LIN {X 0,Y 483.162,Z 602.716,A -85,B 0,C 180,E1 -6752.605,E2 -6752.605} C_VEL
LIN {X 0,Y 482.874,Z 611.081,A -85,B 0,C 180,E1 -6753.546,E2 -6753.546} C_VEL
LIN {X 0,Y 482.488,Z 618.843,A -85,B 0,C 180,E1 -6754.594,E2 -6754.594} C_VEL
LIN {X 0,Y 482.235,Z 626.404,A -85,B 0,C 180,E1 -6755.854,E2 -6755.854} C_VEL
LIN {X 0,Y 481.962,Z 632.514,A -85,B 0,C 180,E1 -6757.125,E2 -6757.125} C_VEL
LIN {X 0,Y 481.753,Z 637.329,A -85,B 0,C 180,E1 -6758.388,E2 -6758.388} C_VEL
LIN {X 0,Y 481.542,Z 641.081,A -85,B 0,C 180,E1 -6759.661,E2 -6759.661} C_VEL
LIN {X 0,Y 481.419,Z 643.812,A -85,B 0,C 180,E1 -6760.939,E2 -6760.939} C_VEL
LIN {X 0,Y 481.414,Z 645.378,A -85,B 0,C 180,E1 -6762.012,E2 -6762.012} C_VEL
LIN {X 0,Y 481.342,Z 646.455,A -85,B 0,C 180,E1 -6763.509,E2 -6763.509} C_VEL
LIN {X 0,Y 481.387,Z 646.173,A -85,B 0,C 180,E1 -6765.235,E2 -6765.235} C_VEL
LIN {X 0,Y 481.377,Z 645.433,A -85,B 0,C 180,E1 -6766.104,E2 -6766.104} C_VEL
LIN {X 0,Y 481.429,Z 644.224,A -85,B 0,C 180,E1 -6766.975,E2 -6766.975} C_VEL
LIN {X 0,Y 481.589,Z 641.181,A -85,B 0,C 180,E1 -6768.457,E2 -6768.457} C_VEL
LIN {X 0,Y 481.792,Z 636.402,A -85,B 0,C 180,E1 -6770.047,E2 -6770.047} C_VEL
LIN {X 0,Y 482.078,Z 631.006,A -85,B 0,C 180,E1 -6771.374,E2 -6771.374} C_VEL
LIN {X 0,Y 482.374,Z 624.124,A -85,B 0,C 180,E1 -6772.711,E2 -6772.711} C_VEL
LIN {X 0,Y 482.765,Z 616.715,A -85,B 0,C 180,E1 -6773.867,E2 -6773.867} C_VEL
LIN {X 0,Y 483.101,Z 608.237,A -85,B 0,C 180,E1 -6774.952,E2 -6774.952} C_VEL
LIN {X 0,Y 483.452,Z 598.406,A -85,B 0,C 180,E1 -6775.971,E2 -6775.971} C_VEL
LIN {X 0,Y 483.892,Z 587.565,A -85,B 0,C 180,E1 -6776.871,E2 -6776.871} C_VEL
LIN {X 0,Y 484.235,Z 576.341,A -85,B 0,C 180,E1 -6777.61,E2 -6777.61} C_VEL
LIN {X 0,Y 484.067,Z 572.549,A -85,B 0,C 180,E1 -6777.827,E2 -6777.827} C_VEL
LIN {X 0,Y 481.719,Z 564.483,A -85,B 0,C 180,E1 -6778.333,E2 -6778.333} C_VEL
LIN {X 0,Y 481.643,Z 564.489,A -85,B 0,C 180,E1 -6781.687,E2 -6781.687} C_VEL
LIN {X 0,Y 481.685,Z 564.485,A -85,B 0,C 180,E1 -6784.681,E2 -6784.681} C_VEL
LIN {X 0,Y 481.655,Z 564.49,A -85,B 0,C 180,E1 -6788.008,E2 -6788.008} C_VEL
LIN {X 0,Y 481.76,Z 564.652,A -85,B 0,C 180,E1 -6790.063,E2 -6790.063} C_VEL
LIN {X 0,Y 482.299,Z 569.987,A -85,B 0,C 180,E1 -6792.089,E2 -6792.089} C_VEL
LIN {X 0,Y 482.189,Z 577.722,A -85,B 0,C 180,E1 -6795.018,E2 -6795.018} C_VEL
LIN {X 0,Y 482.112,Z 585.89,A -85,B 0,C 180,E1 -6798.025,E2 -6798.025} C_VEL
LIN {X 0,Y 481.911,Z 594.241,A -85,B 0,C 180,E1 -6801.164,E2 -6801.164} C_VEL
LIN {X 0,Y 481.765,Z 602.576,A -85,B 0,C 180,E1 -6804.302,E2 -6804.302} C_VEL
LIN {X 0,Y 481.644,Z 610.581,A -85,B 0,C 180,E1 -6807.324,E2 -6807.324} C_VEL
LIN {X 0,Y 481.461,Z 618.342,A -85,B 0,C 180,E1 -6810.244,E2 -6810.244} C_VEL
LIN {X 0,Y 481.363,Z 623.373,A -85,B 0,C 180,E1 -6812.133,E2 -6812.133} C_VEL
LIN {X 0,Y 483.918,Z 637.058,A -85,B 0,C 180,E1 -6812.586,E2 -6812.586} C_VEL
LIN {X 0,Y 483.654,Z 649.638,A -85,B 0,C 180,E1 -6813.085,E2 -6813.085} C_VEL
LIN {X 0,Y 483.238,Z 662.401,A -85,B 0,C 180,E1 -6813.784,E2 -6813.784} C_VEL
LIN {X 0,Y 482.867,Z 673.508,A -85,B 0,C 180,E1 -6814.571,E2 -6814.571} C_VEL
LIN {X 0,Y 482.439,Z 683.68,A -85,B 0,C 180,E1 -6815.47,E2 -6815.47} C_VEL
LIN {X 0,Y 482.016,Z 694.049,A -85,B 0,C 180,E1 -6816.613,E2 -6816.613} C_VEL
LIN {X 0,Y 481.645,Z 702.132,A -85,B 0,C 180,E1 -6817.705,E2 -6817.705} C_VEL
LIN {X 0,Y 481.37,Z 709.469,A -85,B 0,C 180,E1 -6818.921,E2 -6818.921} C_VEL
LIN {X 0,Y 481.161,Z 716.363,A -85,B 0,C 180,E1 -6820.37,E2 -6820.37} C_VEL
LIN {X 0,Y 480.998,Z 721.451,A -85,B 0,C 180,E1 -6821.752,E2 -6821.752} C_VEL
LIN {X 0,Y 480.857,Z 724.91,A -85,B 0,C 180,E1 -6823.004,E2 -6823.004} C_VEL
LIN {X 0,Y 480.806,Z 726.732,A -85,B 0,C 180,E1 -6823.876,E2 -6823.876} C_VEL
LIN {X 0,Y 480.797,Z 728.085,A -85,B 0,C 180,E1 -6824.746,E2 -6824.746} C_VEL
LIN {X 0,Y 480.787,Z 729.027,A -85,B 0,C 180,E1 -6825.612,E2 -6825.612} C_VEL
LIN {X 0,Y 480.739,Z 729.53,A -85,B 0,C 180,E1 -6826.473,E2 -6826.473} C_VEL
LIN {X 0,Y 480.756,Z 729.594,A -85,B 0,C 180,E1 -6827.334,E2 -6827.334} C_VEL
LIN {X 0,Y 480.841,Z 729.198,A -85,B 0,C 180,E1 -6828.309,E2 -6828.309} C_VEL
LIN {X 0,Y 480.833,Z 727.348,A -85,B 0,C 180,E1 -6829.899,E2 -6829.899} C_VEL
LIN {X 0,Y 480.909,Z 724.804,A -85,B 0,C 180,E1 -6831.174,E2 -6831.174} C_VEL
LIN {X 0,Y 481.041,Z 721.245,A -85,B 0,C 180,E1 -6832.445,E2 -6832.445} C_VEL
LIN {X 0,Y 481.163,Z 715.912,A -85,B 0,C 180,E1 -6833.873,E2 -6833.873} C_VEL
LIN {X 0,Y 481.336,Z 709.617,A -85,B 0,C 180,E1 -6835.184,E2 -6835.184} C_VEL
LIN {X 0,Y 481.658,Z 701.976,A -85,B 0,C 180,E1 -6836.445,E2 -6836.445} C_VEL
LIN {X 0,Y 482.063,Z 692.502,A -85,B 0,C 180,E1 -6837.703,E2 -6837.703} C_VEL
LIN {X 0,Y 482.511,Z 682.637,A -85,B 0,C 180,E1 -6838.748,E2 -6838.748} C_VEL
LIN {X 0,Y 482.943,Z 671.629,A -85,B 0,C 180,E1 -6839.688,E2 -6839.688} C_VEL
LIN {X 0,Y 483.344,Z 660.923,A -85,B 0,C 180,E1 -6840.417,E2 -6840.417} C_VEL
LIN {X 0,Y 483.769,Z 649.032,A -85,B 0,C 180,E1 -6841.041,E2 -6841.041} C_VEL
LIN {X 0,Y 483.89,Z 636.377,A -85,B 0,C 180,E1 -6841.535,E2 -6841.535} C_VEL
LIN {X 0,Y 481.718,Z 625.568,A -85,B 0,C 180,E1 -6841.895,E2 -6841.895} C_VEL
LIN {X 0,Y 481.47,Z 624.18,A -85,B 0,C 180,E1 -6841.935,E2 -6841.935} C_VEL
LIN {X 0,Y 481.677,Z 615.891,A -85,B 0,C 180,E1 -6845.023,E2 -6845.023} C_VEL
LIN {X 0,Y 481.773,Z 606.79,A -85,B 0,C 180,E1 -6848.388,E2 -6848.388} C_VEL
LIN {X 0,Y 481.871,Z 599.852,A -85,B 0,C 180,E1 -6850.93,E2 -6850.93} C_VEL
LIN {X 0,Y 481.991,Z 592.674,A -85,B 0,C 180,E1 -6853.492,E2 -6853.492} C_VEL
LIN {X 0,Y 482.013,Z 583.839,A -85,B 0,C 180,E1 -6856.519,E2 -6856.519} C_VEL
LIN {X 0,Y 482.005,Z 574.554,A -85,B 0,C 180,E1 -6859.595,E2 -6859.595} C_VEL
LIN {X 0,Y 481.898,Z 566.032,A -85,B 0,C 180,E1 -6862.283,E2 -6862.283} C_VEL
LIN {X 0,Y 481.683,Z 564.488,A -85,B 0,C 180,E1 -6862.802,E2 -6862.802} C_VEL
LIN {X 0,Y 481.7,Z 564.488,A -85,B 0,C 180,E1 -6865.958,E2 -6865.958} C_VEL
LIN {X 0,Y 481.701,Z 564.485,A -85,B 0,C 180,E1 -6868.782,E2 -6868.782} C_VEL
LIN {X 0,Y 481.654,Z 564.492,A -85,B 0,C 180,E1 -6872.191,E2 -6872.191} C_VEL
LIN {X 0,Y 481.688,Z 564.487,A -85,B 0,C 180,E1 -6874.683,E2 -6874.683} C_VEL
LIN {X 0,Y 481.654,Z 564.49,A -85,B 0,C 180,E1 -6878.009,E2 -6878.009} C_VEL
LIN {X 0,Y 481.681,Z 564.488,A -85,B 0,C 180,E1 -6880.651,E2 -6880.651} C_VEL
LIN {X 0,Y 481.68,Z 564.487,A -85,B 0,C 180,E1 -6883.296,E2 -6883.296} C_VEL
LIN {X 0,Y 481.686,Z 564.486,A -85,B 0,C 180,E1 -6886.847,E2 -6886.847} C_VEL
LIN {X 0,Y 481.741,Z 564.602,A -85,B 0,C 180,E1 -6889.871,E2 -6889.871} C_VEL
LIN {X 0,Y 483.91,Z 575.619,A -85,B 0,C 180,E1 -6893.015,E2 -6893.015} C_VEL
LIN {X 0,Y 484.216,Z 579.325,A -85,B 0,C 180,E1 -6893.99,E2 -6893.99} C_VEL
LIN {X 0,Y 483.665,Z 591.413,A -85,B 0,C 180,E1 -6896.984,E2 -6896.984} C_VEL
LIN {X 0,Y 483.156,Z 605.658,A -85,B 0,C 180,E1 -6900.36,E2 -6900.36} C_VEL
LIN {X 0,Y 482.7,Z 620.019,A -85,B 0,C 180,E1 -6903.637,E2 -6903.637} C_VEL
LIN {X 0,Y 482.294,Z 634.452,A -85,B 0,C 180,E1 -6906.832,E2 -6906.832} C_VEL
LIN {X 0,Y 481.964,Z 648.924,A -85,B 0,C 180,E1 -6909.961,E2 -6909.961} C_VEL
LIN {X 0,Y 481.681,Z 663.387,A -85,B 0,C 180,E1 -6913.035,E2 -6913.035} C_VEL
LIN {X 0,Y 481.527,Z 672.733,A -85,B 0,C 180,E1 -6915.013,E2 -6915.013} C_VEL
LIN {X 0,Y 482.885,Z 686.464,A -85,B 0,C 180,E1 -6915.368,E2 -6915.368} C_VEL
LIN {X 0,Y 483.795,Z 694.327,A -85,B 0,C 180,E1 -6915.65,E2 -6915.65} C_VEL
LIN {X 0,Y 483.332,Z 706.466,A -85,B 0,C 180,E1 -6916.173,E2 -6916.173} C_VEL
LIN {X 0,Y 482.877,Z 718.803,A -85,B 0,C 180,E1 -6916.888,E2 -6916.888} C_VEL
LIN {X 0,Y 482.506,Z 729.607,A -85,B 0,C 180,E1 -6917.685,E2 -6917.685} C_VEL
LIN {X 0,Y 482.04,Z 740.179,A -85,B 0,C 180,E1 -6918.649,E2 -6918.649} C_VEL
LIN {X 0,Y 481.684,Z 749.542,A -85,B 0,C 180,E1 -6919.705,E2 -6919.705} C_VEL
LIN {X 0,Y 481.423,Z 758.694,A -85,B 0,C 180,E1 -6920.972,E2 -6920.972} C_VEL
LIN {X 0,Y 481.209,Z 766.056,A -85,B 0,C 180,E1 -6922.237,E2 -6922.237} C_VEL
LIN {X 0,Y 481.063,Z 772.846,A -85,B 0,C 180,E1 -6923.712,E2 -6923.712} C_VEL
LIN {X 0,Y 481.013,Z 777.288,A -85,B 0,C 180,E1 -6924.972,E2 -6924.972} C_VEL
LIN {X 0,Y 480.986,Z 779.659,A -85,B 0,C 180,E1 -6925.811,E2 -6925.811} C_VEL
LIN {X 0,Y 480.985,Z 781.572,A -85,B 0,C 180,E1 -6926.65,E2 -6926.65} C_VEL
LIN {X 0,Y 480.949,Z 783.04,A -85,B 0,C 180,E1 -6927.488,E2 -6927.488} C_VEL
LIN {X 0,Y 480.93,Z 784.074,A -85,B 0,C 180,E1 -6928.326,E2 -6928.326} C_VEL
LIN {X 0,Y 480.898,Z 784.693,A -85,B 0,C 180,E1 -6929.163,E2 -6929.163} C_VEL
LIN {X 0,Y 480.892,Z 784.904,A -85,B 0,C 180,E1 -6930.001,E2 -6930.001} C_VEL
LIN {X 0,Y 480.898,Z 784.69,A -85,B 0,C 180,E1 -6930.838,E2 -6930.838} C_VEL
LIN {X 0,Y 480.932,Z 784.059,A -85,B 0,C 180,E1 -6931.676,E2 -6931.676} C_VEL
LIN {X 0,Y 480.952,Z 783.019,A -85,B 0,C 180,E1 -6932.513,E2 -6932.513} C_VEL
LIN {X 0,Y 480.986,Z 781.569,A -85,B 0,C 180,E1 -6933.351,E2 -6933.351} C_VEL
LIN {X 0,Y 480.975,Z 778.572,A -85,B 0,C 180,E1 -6934.61,E2 -6934.61} C_VEL
LIN {X 0,Y 481.087,Z 774.505,A -85,B 0,C 180,E1 -6935.87,E2 -6935.87} C_VEL
LIN {X 0,Y 481.154,Z 768.267,A -85,B 0,C 180,E1 -6937.344,E2 -6937.344} C_VEL
LIN {X 0,Y 481.364,Z 761.397,A -85,B 0,C 180,E1 -6938.607,E2 -6938.607} C_VEL
LIN {X 0,Y 481.576,Z 752.955,A -85,B 0,C 180,E1 -6939.874,E2 -6939.874} C_VEL
LIN {X 0,Y 481.917,Z 744.301,A -85,B 0,C 180,E1 -6940.929,E2 -6940.929} C_VEL
LIN {X 0,Y 482.396,Z 733.747,A -85,B 0,C 180,E1 -6941.974,E2 -6941.974} C_VEL
LIN {X 0,Y 482.702,Z 723.405,A -85,B 0,C 180,E1 -6942.808,E2 -6942.808} C_VEL
LIN {X 0,Y 483.164,Z 711.61,A -85,B 0,C 180,E1 -6943.566,E2 -6943.566} C_VEL
LIN {X 0,Y 483.566,Z 699.818,A -85,B 0,C 180,E1 -6944.144,E2 -6944.144} C_VEL
LIN {X 0,Y 483.631,Z 691.789,A -85,B 0,C 180,E1 -6944.451,E2 -6944.451} C_VEL
LIN {X 0,Y 482.182,Z 680.276,A -85,B 0,C 180,E1 -6944.819,E2 -6944.819} C_VEL
LIN {X 0,Y 481.535,Z 673.024,A -85,B 0,C 180,E1 -6944.988,E2 -6944.988} C_VEL
LIN {X 0,Y 481.833,Z 657.99,A -85,B 0,C 180,E1 -6948.193,E2 -6948.193} C_VEL
LIN {X 0,Y 482.121,Z 643.287,A -85,B 0,C 180,E1 -6951.373,E2 -6951.373} C_VEL
LIN {X 0,Y 482.454,Z 629.918,A -85,B 0,C 180,E1 -6954.301,E2 -6954.301} C_VEL
LIN {X 0,Y 482.857,Z 616.074,A -85,B 0,C 180,E1 -6957.394,E2 -6957.394} C_VEL
LIN {X 0,Y 483.243,Z 603.092,A -85,B 0,C 180,E1 -6960.357,E2 -6960.357} C_VEL
LIN {X 0,Y 483.675,Z 590.668,A -85,B 0,C 180,E1 -6963.266,E2 -6963.266} C_VEL
LIN {X 0,Y 484.095,Z 578.209,A -85,B 0,C 180,E1 -6966.271,E2 -6966.271} C_VEL
LIN {X 0,Y 483.339,Z 572.934,A -85,B 0,C 180,E1 -6967.641,E2 -6967.641} C_VEL
LIN {X 0,Y 481.704,Z 564.485,A -85,B 0,C 180,E1 -6969.938,E2 -6969.938} C_VEL
LIN {X 0,Y 481.644,Z 564.493,A -85,B 0,C 180,E1 -6973.3,E2 -6973.3} C_VEL
LIN {X 0,Y 481.663,Z 564.49,A -85,B 0,C 180,E1 -6975.641,E2 -6975.641} C_VEL
LIN {X 0,Y 481.661,Z 564.49,A -85,B 0,C 180,E1 -6978.958,E2 -6978.958} C_VEL
LIN {X 0,Y 481.66,Z 564.489,A -85,B 0,C 180,E1 -6981.993,E2 -6981.993} C_VEL
LIN {X 0,Y 481.698,Z 564.483,A -85,B 0,C 180,E1 -6985.318,E2 -6985.318} C_VEL
LIN {X 0,Y 481.649,Z 564.492,A -85,B 0,C 180,E1 -6988.312,E2 -6988.312} C_VEL
LIN {X 0,Y 481.705,Z 564.481,A -85,B 0,C 180,E1 -6991.219,E2 -6991.219} C_VEL
LIN {X 0,Y 481.705,Z 564.483,A -85,B 0,C 180,E1 -6994.043,E2 -6994.043} C_VEL
LIN {X 0,Y 481.679,Z 564.486,A -85,B 0,C 180,E1 -6996.812,E2 -6996.812} C_VEL
LIN {X 0,Y 481.7,Z 564.482,A -85,B 0,C 180,E1 -6999.503,E2 -6999.503} C_VEL
LIN {X 0,Y 481.712,Z 564.483,A -85,B 0,C 180,E1 -7002.158,E2 -7002.158} C_VEL
LIN {X 0,Y 481.747,Z 564.479,A -85,B 0,C 180,E1 -7004.776,E2 -7004.776} C_VEL
LIN {X 0,Y 481.755,Z 564.478,A -85,B 0,C 180,E1 -7008.215,E2 -7008.215} C_VEL
LIN {X 0,Y 481.767,Z 564.474,A -85,B 0,C 180,E1 -7011.611,E2 -7011.611} C_VEL
LIN {X 0,Y 481.82,Z 564.47,A -85,B 0,C 180,E1 -7014.139,E2 -7014.139} C_VEL
LIN {X 0,Y 481.93,Z 564.454,A -85,B 0,C 180,E1 -7017.492,E2 -7017.492} C_VEL
LIN {X 0,Y 481.91,Z 564.459,A -85,B 0,C 180,E1 -7020.835,E2 -7020.835} C_VEL
LIN {X 0,Y 481.93,Z 564.456,A -85,B 0,C 180,E1 -7022.507,E2 -7022.507} C_VEL
LIN {X 0,Y 481.82,Z 564.469,A -85,B 0,C 180,E1 -7025.86,E2 -7025.86} C_VEL
LIN {X 0,Y 481.766,Z 564.477,A -85,B 0,C 180,E1 -7028.388,E2 -7028.388} C_VEL
LIN {X 0,Y 481.754,Z 564.477,A -85,B 0,C 180,E1 -7031.784,E2 -7031.784} C_VEL
LIN {X 0,Y 481.746,Z 564.478,A -85,B 0,C 180,E1 -7035.224,E2 -7035.224} C_VEL
LIN {X 0,Y 481.715,Z 564.483,A -85,B 0,C 180,E1 -7038.721,E2 -7038.721} C_VEL
LIN {X 0,Y 481.649,Z 564.489,A -85,B 0,C 180,E1 -7041.394,E2 -7041.394} C_VEL
LIN {X 0,Y 481.68,Z 564.486,A -85,B 0,C 180,E1 -7044.113,E2 -7044.113} C_VEL
LIN {X 0,Y 481.749,Z 564.476,A -85,B 0,C 180,E1 -7047.139,E2 -7047.139} C_VEL
LIN {X 0,Y 481.681,Z 564.485,A -85,B 0,C 180,E1 -7049.741,E2 -7049.741} C_VEL
LIN {X 0,Y 481.674,Z 564.489,A -85,B 0,C 180,E1 -7052.674,E2 -7052.674} C_VEL
LIN {X 0,Y 481.645,Z 564.489,A -85,B 0,C 180,E1 -7055.708,E2 -7055.708} C_VEL
LIN {X 0,Y 481.673,Z 564.487,A -85,B 0,C 180,E1 -7058.858,E2 -7058.858} C_VEL
LIN {X 0,Y 481.664,Z 564.487,A -85,B 0,C 180,E1 -7061.914,E2 -7061.914} C_VEL
LIN {X 0,Y 481.661,Z 564.491,A -85,B 0,C 180,E1 -7064.457,E2 -7064.457} C_VEL
LIN {X 0,Y 481.655,Z 564.489,A -85,B 0,C 180,E1 -7067.839,E2 -7067.839} C_VEL
LIN {X 0,Y 481.682,Z 564.487,A -85,B 0,C 180,E1 -7070.65,E2 -7070.65} C_VEL
LIN {X 0,Y 481.628,Z 564.492,A -85,B 0,C 180,E1 -7073.376,E2 -7073.376} C_VEL
LIN {X 0,Y 481.71,Z 564.484,A -85,B 0,C 180,E1 -7076.329,E2 -7076.329} C_VEL
LIN {X 0,Y 481.652,Z 564.489,A -85,B 0,C 180,E1 -7079.417,E2 -7079.417} C_VEL
LIN {X 0,Y 481.701,Z 564.485,A -85,B 0,C 180,E1 -7082.167,E2 -7082.167} C_VEL
LIN {X 0,Y 481.719,Z 564.482,A -85,B 0,C 180,E1 -7084.969,E2 -7084.969} C_VEL
LIN {X 0,Y 481.637,Z 564.49,A -85,B 0,C 180,E1 -7087.981,E2 -7087.981} C_VEL
LIN {X 0,Y 480.97,Z 564.576,A -85,B 0,C 180,E1 -7088.679,E2 -7088.679} C_VEL
LIN {X 0,Y 478.142,Z 564.925,A -85,B 0,C 180,E1 -7089.813,E2 -7089.813} C_VEL
LIN {X 0,Y 475.757,Z 565.225,A -85,B 0,C 180,E1 -7090.727,E2 -7090.727} C_VEL
LIN {X 0,Y 474.737,Z 565.35,A -85,B 0,C 180,E1 -7091.433,E2 -7091.433} C_VEL
LIN {X 0,Y 474.655,Z 565.36,A -85,B 0,C 180,E1 -7091.672,E2 -7091.672} C_VEL
LIN {X 0,Y 474.7,Z 565.357,A -85,B 0,C 180,E1 -7094.544,E2 -7094.544} C_VEL
LIN {X 0,Y 474.739,Z 565.35,A -85,B 0,C 180,E1 -7098.038,E2 -7098.038} C_VEL
LIN {X 0,Y 474.727,Z 565.352,A -85,B 0,C 180,E1 -7101.486,E2 -7101.486} C_VEL
LIN {X 0,Y 474.779,Z 565.346,A -85,B 0,C 180,E1 -7104.052,E2 -7104.052} C_VEL
LIN {X 0,Y 474.895,Z 565.333,A -85,B 0,C 180,E1 -7107.455,E2 -7107.455} C_VEL
LIN {X 0,Y 474.898,Z 565.381,A -85,B 0,C 180,E1 -7109.655,E2 -7109.655} C_VEL
LIN {X 0,Y 477.267,Z 574.753,A -85,B 0,C 180,E1 -7110.21,E2 -7110.21} C_VEL
LIN {X 0,Y 477.003,Z 586.419,A -85,B 0,C 180,E1 -7110.949,E2 -7110.949} C_VEL
LIN {X 0,Y 476.584,Z 596.917,A -85,B 0,C 180,E1 -7111.795,E2 -7111.795} C_VEL
LIN {X 0,Y 476.161,Z 606.491,A -85,B 0,C 180,E1 -7112.749,E2 -7112.749} C_VEL
LIN {X 0,Y 475.822,Z 615.19,A -85,B 0,C 180,E1 -7113.81,E2 -7113.81} C_VEL
LIN {X 0,Y 475.431,Z 623.719,A -85,B 0,C 180,E1 -7115.088,E2 -7115.088} C_VEL
LIN {X 0,Y 475.143,Z 630.521,A -85,B 0,C 180,E1 -7116.368,E2 -7116.368} C_VEL
LIN {X 0,Y 474.878,Z 635.986,A -85,B 0,C 180,E1 -7117.653,E2 -7117.653} C_VEL
LIN {X 0,Y 474.648,Z 640.29,A -85,B 0,C 180,E1 -7118.943,E2 -7118.943} C_VEL
LIN {X 0,Y 474.476,Z 643.537,A -85,B 0,C 180,E1 -7120.238,E2 -7120.238} C_VEL
LIN {X 0,Y 474.397,Z 645.152,A -85,B 0,C 180,E1 -7121.103,E2 -7121.103} C_VEL
LIN {X 0,Y 474.403,Z 646.504,A -85,B 0,C 180,E1 -7122.111,E2 -7122.111} C_VEL
LIN {X 0,Y 474.322,Z 647.506,A -85,B 0,C 180,E1 -7123.713,E2 -7123.713} C_VEL
LIN {X 0,Y 474.32,Z 647.491,A -85,B 0,C 180,E1 -7124.588,E2 -7124.588} C_VEL
LIN {X 0,Y 474.356,Z 646.921,A -85,B 0,C 180,E1 -7125.629,E2 -7125.629} C_VEL
LIN {X 0,Y 474.428,Z 644.907,A -85,B 0,C 180,E1 -7127.233,E2 -7127.233} C_VEL
LIN {X 0,Y 474.607,Z 642.014,A -85,B 0,C 180,E1 -7128.611,E2 -7128.611} C_VEL
LIN {X 0,Y 474.789,Z 638.245,A -85,B 0,C 180,E1 -7129.904,E2 -7129.904} C_VEL
LIN {X 0,Y 475.092,Z 633.08,A -85,B 0,C 180,E1 -7131.26,E2 -7131.26} C_VEL
LIN {X 0,Y 475.411,Z 626.525,A -85,B 0,C 180,E1 -7132.603,E2 -7132.603} C_VEL
LIN {X 0,Y 475.845,Z 618.097,A -85,B 0,C 180,E1 -7133.971,E2 -7133.971} C_VEL
LIN {X 0,Y 476.217,Z 609.43,A -85,B 0,C 180,E1 -7135.105,E2 -7135.105} C_VEL
LIN {X 0,Y 476.591,Z 600.398,A -85,B 0,C 180,E1 -7136.066,E2 -7136.066} C_VEL
LIN {X 0,Y 477.039,Z 590.314,A -85,B 0,C 180,E1 -7136.937,E2 -7136.937} C_VEL
LIN {X 0,Y 477.423,Z 578.333,A -85,B 0,C 180,E1 -7137.76,E2 -7137.76} C_VEL
LIN {X 0,Y 477.153,Z 573.823,A -85,B 0,C 180,E1 -7138.031,E2 -7138.031} C_VEL
LIN {X 0,Y 474.648,Z 565.363,A -85,B 0,C 180,E1 -7138.552,E2 -7138.552} C_VEL
LIN {X 0,Y 474.597,Z 565.365,A -85,B 0,C 180,E1 -7141.217,E2 -7141.217} C_VEL
LIN {X 0,Y 474.627,Z 565.365,A -85,B 0,C 180,E1 -7144.24,E2 -7144.24} C_VEL
LIN {X 0,Y 474.588,Z 565.372,A -85,B 0,C 180,E1 -7147.383,E2 -7147.383} C_VEL
LIN {X 0,Y 474.702,Z 565.368,A -85,B 0,C 180,E1 -7149.846,E2 -7149.846} C_VEL
LIN {X 0,Y 475.291,Z 570.201,A -85,B 0,C 180,E1 -7151.712,E2 -7151.712} C_VEL
LIN {X 0,Y 475.197,Z 578.319,A -85,B 0,C 180,E1 -7154.773,E2 -7154.773} C_VEL
LIN {X 0,Y 475.108,Z 586.118,A -85,B 0,C 180,E1 -7157.697,E2 -7157.697} C_VEL
LIN {X 0,Y 474.902,Z 593.511,A -85,B 0,C 180,E1 -7160.48,E2 -7160.48} C_VEL
LIN {X 0,Y 474.8,Z 601.978,A -85,B 0,C 180,E1 -7163.696,E2 -7163.696} C_VEL
LIN {X 0,Y 474.66,Z 610.123,A -85,B 0,C 180,E1 -7166.782,E2 -7166.782} C_VEL
LIN {X 0,Y 474.433,Z 619.285,A -85,B 0,C 180,E1 -7170.248,E2 -7170.248} C_VEL
LIN {X 0,Y 474.33,Z 623.695,A -85,B 0,C 180,E1 -7171.914,E2 -7171.914} C_VEL
LIN {X 0,Y 476.801,Z 636.577,A -85,B 0,C 180,E1 -7172.344,E2 -7172.344} C_VEL
LIN {X 0,Y 477.076,Z 640.152,A -85,B 0,C 180,E1 -7172.477,E2 -7172.477} C_VEL
LIN {X 0,Y 476.687,Z 653.029,A -85,B 0,C 180,E1 -7173.041,E2 -7173.041} C_VEL
LIN {X 0,Y 476.313,Z 664.755,A -85,B 0,C 180,E1 -7173.727,E2 -7173.727} C_VEL
LIN {X 0,Y 475.842,Z 675.406,A -85,B 0,C 180,E1 -7174.522,E2 -7174.522} C_VEL
LIN {X 0,Y 475.384,Z 686.352,A -85,B 0,C 180,E1 -7175.547,E2 -7175.547} C_VEL
LIN {X 0,Y 474.969,Z 695.819,A -85,B 0,C 180,E1 -7176.642,E2 -7176.642} C_VEL
LIN {X 0,Y 474.561,Z 704.029,A -85,B 0,C 180,E1 -7177.813,E2 -7177.813} C_VEL
LIN {X 0,Y 474.265,Z 711.679,A -85,B 0,C 180,E1 -7179.167,E2 -7179.167} C_VEL
LIN {X 0,Y 474.082,Z 717.731,A -85,B 0,C 180,E1 -7180.516,E2 -7180.516} C_VEL
LIN {X 0,Y 473.916,Z 722.38,A -85,B 0,C 180,E1 -7181.855,E2 -7181.855} C_VEL
LIN {X 0,Y 473.806,Z 724.794,A -85,B 0,C 180,E1 -7182.743,E2 -7182.743} C_VEL
LIN {X 0,Y 473.751,Z 726.753,A -85,B 0,C 180,E1 -7183.629,E2 -7183.629} C_VEL
LIN {X 0,Y 473.711,Z 728.398,A -85,B 0,C 180,E1 -7184.649,E2 -7184.649} C_VEL
LIN {X 0,Y 473.656,Z 729.857,A -85,B 0,C 180,E1 -7186.267,E2 -7186.267} C_VEL
LIN {X 0,Y 473.663,Z 730.035,A -85,B 0,C 180,E1 -7187.141,E2 -7187.141} C_VEL
LIN {X 0,Y 473.758,Z 729.647,A -85,B 0,C 180,E1 -7188.254,E2 -7188.254} C_VEL
LIN {X 0,Y 473.755,Z 728.078,A -85,B 0,C 180,E1 -7189.746,E2 -7189.746} C_VEL
LIN {X 0,Y 473.78,Z 726.566,A -85,B 0,C 180,E1 -7190.609,E2 -7190.609} C_VEL
LIN {X 0,Y 473.938,Z 723.497,A -85,B 0,C 180,E1 -7191.902,E2 -7191.902} C_VEL
LIN {X 0,Y 474.078,Z 718.876,A -85,B 0,C 180,E1 -7193.326,E2 -7193.326} C_VEL
LIN {X 0,Y 474.248,Z 713.117,A -85,B 0,C 180,E1 -7194.686,E2 -7194.686} C_VEL
LIN {X 0,Y 474.473,Z 706.249,A -85,B 0,C 180,E1 -7195.966,E2 -7195.966} C_VEL
LIN {X 0,Y 474.857,Z 697.698,A -85,B 0,C 180,E1 -7197.243,E2 -7197.243} C_VEL
LIN {X 0,Y 475.274,Z 688.954,A -85,B 0,C 180,E1 -7198.306,E2 -7198.306} C_VEL
LIN {X 0,Y 475.708,Z 679.342,A -85,B 0,C 180,E1 -7199.26,E2 -7199.26} C_VEL
LIN {X 0,Y 476.21,Z 667.325,A -85,B 0,C 180,E1 -7200.212,E2 -7200.212} C_VEL
LIN {X 0,Y 476.679,Z 655.297,A -85,B 0,C 180,E1 -7200.951,E2 -7200.951} C_VEL
LIN {X 0,Y 477.087,Z 642.597,A -85,B 0,C 180,E1 -7201.53,E2 -7201.53} C_VEL
LIN {X 0,Y 476.864,Z 636.22,A -85,B 0,C 180,E1 -7201.769,E2 -7201.769} C_VEL
LIN {X 0,Y 474.421,Z 624.575,A -85,B 0,C 180,E1 -7202.176,E2 -7202.176} C_VEL
LIN {X 0,Y 474.654,Z 616.756,A -85,B 0,C 180,E1 -7205.097,E2 -7205.097} C_VEL
LIN {X 0,Y 474.759,Z 607.573,A -85,B 0,C 180,E1 -7208.513,E2 -7208.513} C_VEL
LIN {X 0,Y 474.957,Z 598.27,A -85,B 0,C 180,E1 -7211.956,E2 -7211.956} C_VEL
LIN {X 0,Y 475,Z 589.518,A -85,B 0,C 180,E1 -7215.007,E2 -7215.007} C_VEL
LIN {X 0,Y 475.005,Z 580.408,A -85,B 0,C 180,E1 -7218.102,E2 -7218.102} C_VEL
LIN {X 0,Y 474.954,Z 572.173,A -85,B 0,C 180,E1 -7220.802,E2 -7220.802} C_VEL
LIN {X 0,Y 474.803,Z 566.401,A -85,B 0,C 180,E1 -7222.635,E2 -7222.635} C_VEL
LIN {X 0,Y 474.634,Z 565.367,A -85,B 0,C 180,E1 -7223.048,E2 -7223.048} C_VEL
LIN {X 0,Y 474.664,Z 565.365,A -85,B 0,C 180,E1 -7225.429,E2 -7225.429} C_VEL
LIN {X 0,Y 474.644,Z 565.364,A -85,B 0,C 180,E1 -7228.283,E2 -7228.283} C_VEL
LIN {X 0,Y 474.597,Z 565.37,A -85,B 0,C 180,E1 -7231.218,E2 -7231.218} C_VEL
LIN {X 0,Y 474.629,Z 565.366,A -85,B 0,C 180,E1 -7234.242,E2 -7234.242} C_VEL
LIN {X 0,Y 474.59,Z 565.371,A -85,B 0,C 180,E1 -7237.384,E2 -7237.384} C_VEL
LIN {X 0,Y 474.646,Z 565.363,A -85,B 0,C 180,E1 -7239.652,E2 -7239.652} C_VEL
LIN {X 0,Y 474.648,Z 565.363,A -85,B 0,C 180,E1 -7242.931,E2 -7242.931} C_VEL
LIN {X 0,Y 474.615,Z 565.367,A -85,B 0,C 180,E1 -7245.897,E2 -7245.897} C_VEL
LIN {X 0,Y 474.642,Z 565.367,A -85,B 0,C 180,E1 -7249.039,E2 -7249.039} C_VEL
LIN {X 0,Y 474.687,Z 565.48,A -85,B 0,C 180,E1 -7249.538,E2 -7249.538} C_VEL
LIN {X 0,Y 476.849,Z 576.438,A -85,B 0,C 180,E1 -7252.738,E2 -7252.738} C_VEL
LIN {X 0,Y 477.289,Z 580.764,A -85,B 0,C 180,E1 -7253.916,E2 -7253.916} C_VEL
LIN {X 0,Y 476.696,Z 592.809,A -85,B 0,C 180,E1 -7256.943,E2 -7256.943} C_VEL
LIN {X 0,Y 476.169,Z 606.581,A -85,B 0,C 180,E1 -7260.274,E2 -7260.274} C_VEL
LIN {X 0,Y 475.68,Z 620.245,A -85,B 0,C 180,E1 -7263.454,E2 -7263.454} C_VEL
LIN {X 0,Y 475.248,Z 634.618,A -85,B 0,C 180,E1 -7266.699,E2 -7266.699} C_VEL
LIN {X 0,Y 474.884,Z 648.998,A -85,B 0,C 180,E1 -7269.875,E2 -7269.875} C_VEL
LIN {X 0,Y 474.621,Z 662.355,A -85,B 0,C 180,E1 -7272.774,E2 -7272.774} C_VEL
LIN {X 0,Y 474.437,Z 671.694,A -85,B 0,C 180,E1 -7274.784,E2 -7274.784} C_VEL
LIN {X 0,Y 475.918,Z 687.18,A -85,B 0,C 180,E1 -7275.202,E2 -7275.202} C_VEL
LIN {X 0,Y 476.827,Z 694.662,A -85,B 0,C 180,E1 -7275.49,E2 -7275.49} C_VEL
LIN {X 0,Y 476.348,Z 706.409,A -85,B 0,C 180,E1 -7276.02,E2 -7276.02} C_VEL
LIN {X 0,Y 475.847,Z 718.863,A -85,B 0,C 180,E1 -7276.767,E2 -7276.767} C_VEL
LIN {X 0,Y 475.468,Z 729.448,A -85,B 0,C 180,E1 -7277.574,E2 -7277.574} C_VEL
LIN {X 0,Y 474.961,Z 740.128,A -85,B 0,C 180,E1 -7278.586,E2 -7278.586} C_VEL
LIN {X 0,Y 474.567,Z 750.155,A -85,B 0,C 180,E1 -7279.764,E2 -7279.764} C_VEL
LIN {X 0,Y 474.312,Z 759.007,A -85,B 0,C 180,E1 -7281.05,E2 -7281.05} C_VEL
LIN {X 0,Y 474.098,Z 767.257,A -85,B 0,C 180,E1 -7282.548,E2 -7282.548} C_VEL
LIN {X 0,Y 473.996,Z 773.655,A -85,B 0,C 180,E1 -7284.043,E2 -7284.043} C_VEL
LIN {X 0,Y 473.901,Z 777.824,A -85,B 0,C 180,E1 -7285.322,E2 -7285.322} C_VEL
LIN {X 0,Y 473.91,Z 780.908,A -85,B 0,C 180,E1 -7286.6,E2 -7286.6} C_VEL
LIN {X 0,Y 473.89,Z 782.399,A -85,B 0,C 180,E1 -7287.451,E2 -7287.451} C_VEL
LIN {X 0,Y 473.857,Z 783.447,A -85,B 0,C 180,E1 -7288.301,E2 -7288.301} C_VEL
LIN {X 0,Y 473.823,Z 784.083,A -85,B 0,C 180,E1 -7289.151,E2 -7289.151} C_VEL
LIN {X 0,Y 473.818,Z 784.304,A -85,B 0,C 180,E1 -7290.001,E2 -7290.001} C_VEL
LIN {X 0,Y 473.822,Z 784.098,A -85,B 0,C 180,E1 -7290.851,E2 -7290.851} C_VEL
LIN {X 0,Y 473.859,Z 783.466,A -85,B 0,C 180,E1 -7291.701,E2 -7291.701} C_VEL
LIN {X 0,Y 473.892,Z 782.428,A -85,B 0,C 180,E1 -7292.551,E2 -7292.551} C_VEL
LIN {X 0,Y 473.91,Z 780.971,A -85,B 0,C 180,E1 -7293.401,E2 -7293.401} C_VEL
LIN {X 0,Y 473.889,Z 777.959,A -85,B 0,C 180,E1 -7294.679,E2 -7294.679} C_VEL
LIN {X 0,Y 474.006,Z 773.864,A -85,B 0,C 180,E1 -7295.958,E2 -7295.958} C_VEL
LIN {X 0,Y 474.07,Z 767.538,A -85,B 0,C 180,E1 -7297.454,E2 -7297.454} C_VEL
LIN {X 0,Y 474.288,Z 760.558,A -85,B 0,C 180,E1 -7298.737,E2 -7298.737} C_VEL
LIN {X 0,Y 474.522,Z 751.93,A -85,B 0,C 180,E1 -7300.023,E2 -7300.023} C_VEL
LIN {X 0,Y 474.905,Z 743.284,A -85,B 0,C 180,E1 -7301.093,E2 -7301.093} C_VEL
LIN {X 0,Y 475.386,Z 733.052,A -85,B 0,C 180,E1 -7302.125,E2 -7302.125} C_VEL
LIN {X 0,Y 475.769,Z 722.104,A -85,B 0,C 180,E1 -7303.019,E2 -7303.019} C_VEL
LIN {X 0,Y 476.244,Z 710.601,A -85,B 0,C 180,E1 -7303.767,E2 -7303.767} C_VEL
LIN {X 0,Y 476.645,Z 698.806,A -85,B 0,C 180,E1 -7304.354,E2 -7304.354} C_VEL
LIN {X 0,Y 476.61,Z 691.914,A -85,B 0,C 180,E1 -7304.627,E2 -7304.627} C_VEL
LIN {X 0,Y 475.255,Z 680.404,A -85,B 0,C 180,E1 -7305.013,E2 -7305.013} C_VEL
LIN {X 0,Y 474.443,Z 671.993,A -85,B 0,C 180,E1 -7305.217,E2 -7305.217} C_VEL
LIN {X 0,Y 474.768,Z 657.447,A -85,B 0,C 180,E1 -7308.39,E2 -7308.39} C_VEL
LIN {X 0,Y 475.059,Z 643.631,A -85,B 0,C 180,E1 -7311.426,E2 -7311.426} C_VEL
LIN {X 0,Y 475.498,Z 627.992,A -85,B 0,C 180,E1 -7314.913,E2 -7314.913} C_VEL
LIN {X 0,Y 475.858,Z 615.086,A -85,B 0,C 180,E1 -7317.858,E2 -7317.858} C_VEL
LIN {X 0,Y 476.259,Z 603.242,A -85,B 0,C 180,E1 -7320.605,E2 -7320.605} C_VEL
LIN {X 0,Y 476.76,Z 590.835,A -85,B 0,C 180,E1 -7323.56,E2 -7323.56} C_VEL
LIN {X 0,Y 477.165,Z 579.458,A -85,B 0,C 180,E1 -7326.359,E2 -7326.359} C_VEL
LIN {X 0,Y 476.142,Z 573.076,A -85,B 0,C 180,E1 -7328.043,E2 -7328.043} C_VEL
LIN {X 0,Y 474.65,Z 565.364,A -85,B 0,C 180,E1 -7330.2,E2 -7330.2} C_VEL
LIN {X 0,Y 474.607,Z 565.369,A -85,B 0,C 180,E1 -7333.481,E2 -7333.481} C_VEL
LIN {X 0,Y 474.607,Z 565.369,A -85,B 0,C 180,E1 -7336.519,E2 -7336.519} C_VEL
LIN {X 0,Y 474.622,Z 565.367,A -85,B 0,C 180,E1 -7339.342,E2 -7339.342} C_VEL
LIN {X 0,Y 474.615,Z 565.367,A -85,B 0,C 180,E1 -7341.704,E2 -7341.704} C_VEL
LIN {X 0,Y 474.635,Z 565.365,A -85,B 0,C 180,E1 -7344.726,E2 -7344.726} C_VEL
LIN {X 0,Y 474.64,Z 565.363,A -85,B 0,C 180,E1 -7347.788,E2 -7347.788} C_VEL
LIN {X 0,Y 474.629,Z 565.364,A -85,B 0,C 180,E1 -7350.885,E2 -7350.885} C_VEL
LIN {X 0,Y 474.665,Z 565.359,A -85,B 0,C 180,E1 -7353.628,E2 -7353.628} C_VEL
LIN {X 0,Y 474.64,Z 565.364,A -85,B 0,C 180,E1 -7356.641,E2 -7356.641} C_VEL
LIN {X 0,Y 474.659,Z 565.362,A -85,B 0,C 180,E1 -7360.089,E2 -7360.089} C_VEL
LIN {X 0,Y 474.655,Z 565.361,A -85,B 0,C 180,E1 -7362.774,E2 -7362.774} C_VEL
LIN {X 0,Y 474.652,Z 565.359,A -85,B 0,C 180,E1 -7365.421,E2 -7365.421} C_VEL
LIN {X 0,Y 474.708,Z 565.355,A -85,B 0,C 180,E1 -7368.037,E2 -7368.037} C_VEL
LIN {X 0,Y 474.732,Z 565.35,A -85,B 0,C 180,E1 -7371.486,E2 -7371.486} C_VEL
LIN {X 0,Y 474.783,Z 565.346,A -85,B 0,C 180,E1 -7374.052,E2 -7374.052} C_VEL
LIN {X 0,Y 474.896,Z 565.33,A -85,B 0,C 180,E1 -7377.455,E2 -7377.455} C_VEL
LIN {X 0,Y 474.916,Z 565.329,A -85,B 0,C 180,E1 -7380,E2 -7380} C_VEL
LIN {X 0,Y 474.896,Z 565.332,A -85,B 0,C 180,E1 -7382.544,E2 -7382.544} C_VEL
LIN {X 0,Y 474.783,Z 565.346,A -85,B 0,C 180,E1 -7385.947,E2 -7385.947} C_VEL
LIN {X 0,Y 474.731,Z 565.353,A -85,B 0,C 180,E1 -7388.513,E2 -7388.513} C_VEL
LIN {X 0,Y 474.707,Z 565.356,A -85,B 0,C 180,E1 -7391.962,E2 -7391.962} C_VEL
LIN {X 0,Y 474.703,Z 565.354,A -85,B 0,C 180,E1 -7395.455,E2 -7395.455} C_VEL
LIN {X 0,Y 474.667,Z 565.359,A -85,B 0,C 180,E1 -7399.01,E2 -7399.01} C_VEL
LIN {X 0,Y 474.593,Z 565.367,A -85,B 0,C 180,E1 -7401.728,E2 -7401.728} C_VEL
LIN {X 0,Y 474.662,Z 565.363,A -85,B 0,C 180,E1 -7404.492,E2 -7404.492} C_VEL
LIN {X 0,Y 474.683,Z 565.355,A -85,B 0,C 180,E1 -7407.334,E2 -7407.334} C_VEL
LIN {X 0,Y 474.607,Z 565.368,A -85,B 0,C 180,E1 -7410.23,E2 -7410.23} C_VEL
LIN {X 0,Y 474.645,Z 565.361,A -85,B 0,C 180,E1 -7413.219,E2 -7413.219} C_VEL
LIN {X 0,Y 474.595,Z 565.371,A -85,B 0,C 180,E1 -7416.323,E2 -7416.323} C_VEL
LIN {X 0,Y 474.629,Z 565.364,A -85,B 0,C 180,E1 -7419.647,E2 -7419.647} C_VEL
LIN {X 0,Y 474.636,Z 565.365,A -85,B 0,C 180,E1 -7422.931,E2 -7422.931} C_VEL
LIN {X 0,Y 474.616,Z 565.367,A -85,B 0,C 180,E1 -7425.895,E2 -7425.895} C_VEL
LIN {X 0,Y 474.633,Z 565.364,A -85,B 0,C 180,E1 -7429.04,E2 -7429.04} C_VEL
LIN {X 0,Y 474.611,Z 565.366,A -85,B 0,C 180,E1 -7431.703,E2 -7431.703} C_VEL
LIN {X 0,Y 474.625,Z 565.367,A -85,B 0,C 180,E1 -7434.725,E2 -7434.725} C_VEL
LIN {X 0,Y 474.638,Z 565.362,A -85,B 0,C 180,E1 -7437.787,E2 -7437.787} C_VEL
LIN {X 0,Y 474.624,Z 565.365,A -85,B 0,C 180,E1 -7440.884,E2 -7440.884} C_VEL
LIN {X 0,Y 474.661,Z 565.359,A -85,B 0,C 180,E1 -7443.628,E2 -7443.628} C_VEL
LIN {X 0,Y 474.636,Z 565.365,A -85,B 0,C 180,E1 -7446.641,E2 -7446.641} C_VEL
LIN {X 0,Y 474.655,Z 565.362,A -85,B 0,C 180,E1 -7450.089,E2 -7450.089} C_VEL
LIN {X 0,Y 474.655,Z 565.36,A -85,B 0,C 180,E1 -7451.672,E2 -7451.672} C_VEL
LIN {X 0,Y 473.993,Z 565.445,A -85,B 0,C 180,E1 -7452.381,E2 -7452.381} C_VEL
LIN {X 0,Y 471.142,Z 565.799,A -85,B 0,C 180,E1 -7453.533,E2 -7453.533} C_VEL
LIN {X 0,Y 468.725,Z 566.101,A -85,B 0,C 180,E1 -7454.461,E2 -7454.461} C_VEL
LIN {X 0,Y 467.684,Z 566.229,A -85,B 0,C 180,E1 -7455.178,E2 -7455.178} C_VEL
LIN {X 0,Y 467.597,Z 566.238,A -85,B 0,C 180,E1 -7455.421,E2 -7455.421} C_VEL
LIN {X 0,Y 467.683,Z 566.228,A -85,B 0,C 180,E1 -7457.855,E2 -7457.855} C_VEL
LIN {X 0,Y 467.681,Z 566.229,A -85,B 0,C 180,E1 -7461.357,E2 -7461.357} C_VEL
LIN {X 0,Y 467.743,Z 566.221,A -85,B 0,C 180,E1 -7463.962,E2 -7463.962} C_VEL
LIN {X 0,Y 467.86,Z 566.209,A -85,B 0,C 180,E1 -7467.416,E2 -7467.416} C_VEL
LIN {X 0,Y 467.857,Z 566.209,A -85,B 0,C 180,E1 -7469.434,E2 -7469.434} C_VEL
LIN {X 0,Y 470.311,Z 575.423,A -85,B 0,C 180,E1 -7469.999,E2 -7469.999} C_VEL
LIN {X 0,Y 470.161,Z 585.584,A -85,B 0,C 180,E1 -7470.642,E2 -7470.642} C_VEL
LIN {X 0,Y 469.792,Z 596.481,A -85,B 0,C 180,E1 -7471.499,E2 -7471.499} C_VEL
LIN {X 0,Y 469.373,Z 605.352,A -85,B 0,C 180,E1 -7472.359,E2 -7472.359} C_VEL
LIN {X 0,Y 468.985,Z 614.449,A -85,B 0,C 180,E1 -7473.436,E2 -7473.436} C_VEL
LIN {X 0,Y 468.509,Z 623.291,A -85,B 0,C 180,E1 -7474.732,E2 -7474.732} C_VEL
LIN {X 0,Y 468.233,Z 630.394,A -85,B 0,C 180,E1 -7476.03,E2 -7476.03} C_VEL
LIN {X 0,Y 467.898,Z 636.9,A -85,B 0,C 180,E1 -7477.547,E2 -7477.547} C_VEL
LIN {X 0,Y 467.624,Z 641.854,A -85,B 0,C 180,E1 -7479.079,E2 -7479.079} C_VEL
LIN {X 0,Y 467.451,Z 644.948,A -85,B 0,C 180,E1 -7480.393,E2 -7480.393} C_VEL
LIN {X 0,Y 467.386,Z 646.487,A -85,B 0,C 180,E1 -7481.272,E2 -7481.272} C_VEL
LIN {X 0,Y 467.366,Z 647.608,A -85,B 0,C 180,E1 -7482.197,E2 -7482.197} C_VEL
LIN {X 0,Y 467.298,Z 648.559,A -85,B 0,C 180,E1 -7483.923,E2 -7483.923} C_VEL
LIN {X 0,Y 467.303,Z 648.454,A -85,B 0,C 180,E1 -7484.812,E2 -7484.812} C_VEL
LIN {X 0,Y 467.334,Z 647.862,A -85,B 0,C 180,E1 -7485.75,E2 -7485.75} C_VEL
LIN {X 0,Y 467.457,Z 645.589,A -85,B 0,C 180,E1 -7487.498,E2 -7487.498} C_VEL
LIN {X 0,Y 467.638,Z 642.838,A -85,B 0,C 180,E1 -7488.773,E2 -7488.773} C_VEL
LIN {X 0,Y 467.871,Z 638.582,A -85,B 0,C 180,E1 -7490.211,E2 -7490.211} C_VEL
LIN {X 0,Y 468.198,Z 632.795,A -85,B 0,C 180,E1 -7491.674,E2 -7491.674} C_VEL
LIN {X 0,Y 468.533,Z 626.399,A -85,B 0,C 180,E1 -7492.953,E2 -7492.953} C_VEL
LIN {X 0,Y 468.95,Z 619.481,A -85,B 0,C 180,E1 -7494.079,E2 -7494.079} C_VEL
LIN {X 0,Y 469.365,Z 610.66,A -85,B 0,C 180,E1 -7495.26,E2 -7495.26} C_VEL
LIN {X 0,Y 469.771,Z 601.11,A -85,B 0,C 180,E1 -7496.291,E2 -7496.291} C_VEL
LIN {X 0,Y 470.261,Z 590.179,A -85,B 0,C 180,E1 -7497.237,E2 -7497.237} C_VEL
LIN {X 0,Y 470.675,Z 578.177,A -85,B 0,C 180,E1 -7498.054,E2 -7498.054} C_VEL
LIN {X 0,Y 470.13,Z 574.661,A -85,B 0,C 180,E1 -7498.278,E2 -7498.278} C_VEL
LIN {X 0,Y 467.596,Z 566.242,A -85,B 0,C 180,E1 -7498.807,E2 -7498.807} C_VEL
LIN {X 0,Y 467.58,Z 566.24,A -85,B 0,C 180,E1 -7501.739,E2 -7501.739} C_VEL
LIN {X 0,Y 467.561,Z 566.245,A -85,B 0,C 180,E1 -7504.832,E2 -7504.832} C_VEL
LIN {X 0,Y 467.566,Z 566.245,A -85,B 0,C 180,E1 -7508.043,E2 -7508.043} C_VEL
LIN {X 0,Y 467.662,Z 566.344,A -85,B 0,C 180,E1 -7509.728,E2 -7509.728} C_VEL
LIN {X 0,Y 468.303,Z 571.891,A -85,B 0,C 180,E1 -7511.898,E2 -7511.898} C_VEL
LIN {X 0,Y 468.207,Z 580.503,A -85,B 0,C 180,E1 -7515.131,E2 -7515.131} C_VEL
LIN {X 0,Y 468.094,Z 588.239,A -85,B 0,C 180,E1 -7518.078,E2 -7518.078} C_VEL
LIN {X 0,Y 467.872,Z 595.652,A -85,B 0,C 180,E1 -7520.885,E2 -7520.885} C_VEL
LIN {X 0,Y 467.778,Z 602.768,A -85,B 0,C 180,E1 -7523.598,E2 -7523.598} C_VEL
LIN {X 0,Y 467.638,Z 610.979,A -85,B 0,C 180,E1 -7526.733,E2 -7526.733} C_VEL
LIN {X 0,Y 467.393,Z 620.229,A -85,B 0,C 180,E1 -7530.251,E2 -7530.251} C_VEL
LIN {X 0,Y 467.297,Z 624.007,A -85,B 0,C 180,E1 -7531.681,E2 -7531.681} C_VEL
LIN {X 0,Y 469.938,Z 637.528,A -85,B 0,C 180,E1 -7532.153,E2 -7532.153} C_VEL
LIN {X 0,Y 470.171,Z 642.048,A -85,B 0,C 180,E1 -7532.329,E2 -7532.329} C_VEL
LIN {X 0,Y 469.734,Z 654.736,A -85,B 0,C 180,E1 -7532.91,E2 -7532.91} C_VEL
LIN {X 0,Y 469.34,Z 666.331,A -85,B 0,C 180,E1 -7533.622,E2 -7533.622} C_VEL
LIN {X 0,Y 468.857,Z 677.227,A -85,B 0,C 180,E1 -7534.472,E2 -7534.472} C_VEL
LIN {X 0,Y 468.351,Z 687.917,A -85,B 0,C 180,E1 -7535.51,E2 -7535.51} C_VEL
LIN {X 0,Y 467.928,Z 697.274,A -85,B 0,C 180,E1 -7536.642,E2 -7536.642} C_VEL
LIN {X 0,Y 467.458,Z 705.872,A -85,B 0,C 180,E1 -7537.923,E2 -7537.923} C_VEL
LIN {X 0,Y 467.202,Z 713.245,A -85,B 0,C 180,E1 -7539.299,E2 -7539.299} C_VEL
LIN {X 0,Y 466.983,Z 719.004,A -85,B 0,C 180,E1 -7540.665,E2 -7540.665} C_VEL
LIN {X 0,Y 466.824,Z 723.449,A -85,B 0,C 180,E1 -7542.024,E2 -7542.024} C_VEL
LIN {X 0,Y 466.696,Z 726.721,A -85,B 0,C 180,E1 -7543.374,E2 -7543.374} C_VEL
LIN {X 0,Y 466.659,Z 728.701,A -85,B 0,C 180,E1 -7544.544,E2 -7544.544} C_VEL
LIN {X 0,Y 466.569,Z 730.145,A -85,B 0,C 180,E1 -7546.054,E2 -7546.054} C_VEL
LIN {X 0,Y 466.566,Z 730.44,A -85,B 0,C 180,E1 -7546.942,E2 -7546.942} C_VEL
LIN {X 0,Y 466.681,Z 730.097,A -85,B 0,C 180,E1 -7548.195,E2 -7548.195} C_VEL
LIN {X 0,Y 466.67,Z 728.751,A -85,B 0,C 180,E1 -7549.589,E2 -7549.589} C_VEL
LIN {X 0,Y 466.689,Z 727.371,A -85,B 0,C 180,E1 -7550.465,E2 -7550.465} C_VEL
LIN {X 0,Y 466.845,Z 724.451,A -85,B 0,C 180,E1 -7551.778,E2 -7551.778} C_VEL
LIN {X 0,Y 467.004,Z 719.625,A -85,B 0,C 180,E1 -7553.324,E2 -7553.324} C_VEL
LIN {X 0,Y 467.218,Z 713.408,A -85,B 0,C 180,E1 -7554.822,E2 -7554.822} C_VEL
LIN {X 0,Y 467.488,Z 706.497,A -85,B 0,C 180,E1 -7556.121,E2 -7556.121} C_VEL
LIN {X 0,Y 467.898,Z 697.918,A -85,B 0,C 180,E1 -7557.418,E2 -7557.418} C_VEL
LIN {X 0,Y 468.338,Z 689.143,A -85,B 0,C 180,E1 -7558.496,E2 -7558.496} C_VEL
LIN {X 0,Y 468.842,Z 678.249,A -85,B 0,C 180,E1 -7559.571,E2 -7559.571} C_VEL
LIN {X 0,Y 469.341,Z 667.39,A -85,B 0,C 180,E1 -7560.429,E2 -7560.429} C_VEL
LIN {X 0,Y 469.821,Z 655.235,A -85,B 0,C 180,E1 -7561.179,E2 -7561.179} C_VEL
LIN {X 0,Y 470.251,Z 642.427,A -85,B 0,C 180,E1 -7561.767,E2 -7561.767} C_VEL
LIN {X 0,Y 469.954,Z 636.81,A -85,B 0,C 180,E1 -7561.982,E2 -7561.982} C_VEL
LIN {X 0,Y 467.333,Z 624.979,A -85,B 0,C 180,E1 -7562.424,E2 -7562.424} C_VEL
LIN {X 0,Y 467.636,Z 617.684,A -85,B 0,C 180,E1 -7565.174,E2 -7565.174} C_VEL
LIN {X 0,Y 467.753,Z 608.361,A -85,B 0,C 180,E1 -7568.642,E2 -7568.642} C_VEL
LIN {X 0,Y 467.937,Z 600.076,A -85,B 0,C 180,E1 -7571.699,E2 -7571.699} C_VEL
LIN {X 0,Y 467.978,Z 592.693,A -85,B 0,C 180,E1 -7574.347,E2 -7574.347} C_VEL
LIN {X 0,Y 468.065,Z 583.612,A -85,B 0,C 180,E1 -7577.476,E2 -7577.476} C_VEL
LIN {X 0,Y 468.042,Z 575.476,A -85,B 0,C 180,E1 -7580.204,E2 -7580.204} C_VEL
LIN {X 0,Y 467.905,Z 568.301,A -85,B 0,C 180,E1 -7582.521,E2 -7582.521} C_VEL
LIN {X 0,Y 467.596,Z 566.244,A -85,B 0,C 180,E1 -7583.238,E2 -7583.238} C_VEL
LIN {X 0,Y 467.605,Z 566.244,A -85,B 0,C 180,E1 -7585.841,E2 -7585.841} C_VEL
LIN {X 0,Y 467.577,Z 566.244,A -85,B 0,C 180,E1 -7588.75,E2 -7588.75} C_VEL
LIN {X 0,Y 467.58,Z 566.244,A -85,B 0,C 180,E1 -7591.741,E2 -7591.741} C_VEL
LIN {X 0,Y 467.564,Z 566.246,A -85,B 0,C 180,E1 -7594.833,E2 -7594.833} C_VEL
LIN {X 0,Y 467.566,Z 566.245,A -85,B 0,C 180,E1 -7598.045,E2 -7598.045} C_VEL
LIN {X 0,Y 467.592,Z 566.241,A -85,B 0,C 180,E1 -7600.264,E2 -7600.264} C_VEL
LIN {X 0,Y 467.615,Z 566.235,A -85,B 0,C 180,E1 -7602.572,E2 -7602.572} C_VEL
LIN {X 0,Y 467.571,Z 566.243,A -85,B 0,C 180,E1 -7606.177,E2 -7606.177} C_VEL
LIN {X 0,Y 467.602,Z 566.278,A -85,B 0,C 180,E1 -7609.173,E2 -7609.173} C_VEL
LIN {X 0,Y 469.26,Z 574.554,A -85,B 0,C 180,E1 -7611.675,E2 -7611.675} C_VEL
LIN {X 0,Y 470.321,Z 580.202,A -85,B 0,C 180,E1 -7613.295,E2 -7613.295} C_VEL
LIN {X 0,Y 470.058,Z 588.142,A -85,B 0,C 180,E1 -7615.38,E2 -7615.38} C_VEL
LIN {X 0,Y 469.397,Z 600.945,A -85,B 0,C 180,E1 -7618.587,E2 -7618.587} C_VEL
LIN {X 0,Y 468.941,Z 612.33,A -85,B 0,C 180,E1 -7621.343,E2 -7621.343} C_VEL
LIN {X 0,Y 468.491,Z 625.584,A -85,B 0,C 180,E1 -7624.452,E2 -7624.452} C_VEL
LIN {X 0,Y 468.069,Z 638.854,A -85,B 0,C 180,E1 -7627.489,E2 -7627.489} C_VEL
LIN {X 0,Y 467.74,Z 653.173,A -85,B 0,C 180,E1 -7630.698,E2 -7630.698} C_VEL
LIN {X 0,Y 467.46,Z 667.686,A -85,B 0,C 180,E1 -7633.897,E2 -7633.897} C_VEL
LIN {X 0,Y 467.361,Z 670.647,A -85,B 0,C 180,E1 -7634.548,E2 -7634.548} C_VEL
LIN {X 0,Y 468.744,Z 685.675,A -85,B 0,C 180,E1 -7634.956,E2 -7634.956} C_VEL
LIN {X 0,Y 469.878,Z 694.916,A -85,B 0,C 180,E1 -7635.326,E2 -7635.326} C_VEL
LIN {X 0,Y 469.355,Z 707.359,A -85,B 0,C 180,E1 -7635.918,E2 -7635.918} C_VEL
LIN {X 0,Y 468.805,Z 719.372,A -85,B 0,C 180,E1 -7636.675,E2 -7636.675} C_VEL
LIN {X 0,Y 468.409,Z 730.379,A -85,B 0,C 180,E1 -7637.563,E2 -7637.563} C_VEL
LIN {X 0,Y 467.882,Z 740.077,A -85,B 0,C 180,E1 -7638.521,E2 -7638.521} C_VEL
LIN {X 0,Y 467.471,Z 750.962,A -85,B 0,C 180,E1 -7639.826,E2 -7639.826} C_VEL
LIN {X 0,Y 467.213,Z 759.757,A -85,B 0,C 180,E1 -7641.131,E2 -7641.131} C_VEL
LIN {X 0,Y 467.019,Z 766.784,A -85,B 0,C 180,E1 -7642.434,E2 -7642.434} C_VEL
LIN {X 0,Y 466.896,Z 773.212,A -85,B 0,C 180,E1 -7643.952,E2 -7643.952} C_VEL
LIN {X 0,Y 466.819,Z 777.396,A -85,B 0,C 180,E1 -7645.251,E2 -7645.251} C_VEL
LIN {X 0,Y 466.837,Z 780.482,A -85,B 0,C 180,E1 -7646.549,E2 -7646.549} C_VEL
LIN {X 0,Y 466.801,Z 781.977,A -85,B 0,C 180,E1 -7647.412,E2 -7647.412} C_VEL
LIN {X 0,Y 466.786,Z 783.028,A -85,B 0,C 180,E1 -7648.275,E2 -7648.275} C_VEL
LIN {X 0,Y 466.747,Z 783.67,A -85,B 0,C 180,E1 -7649.138,E2 -7649.138} C_VEL
LIN {X 0,Y 466.739,Z 783.9,A -85,B 0,C 180,E1 -7650.001,E2 -7650.001} C_VEL
LIN {X 0,Y 466.746,Z 783.7,A -85,B 0,C 180,E1 -7650.864,E2 -7650.864} C_VEL
LIN {X 0,Y 466.788,Z 783.074,A -85,B 0,C 180,E1 -7651.726,E2 -7651.726} C_VEL
LIN {X 0,Y 466.804,Z 782.04,A -85,B 0,C 180,E1 -7652.59,E2 -7652.59} C_VEL
LIN {X 0,Y 466.836,Z 780.582,A -85,B 0,C 180,E1 -7653.453,E2 -7653.453} C_VEL
LIN {X 0,Y 466.808,Z 777.567,A -85,B 0,C 180,E1 -7654.751,E2 -7654.751} C_VEL
LIN {X 0,Y 466.904,Z 773.453,A -85,B 0,C 180,E1 -7656.049,E2 -7656.049} C_VEL
LIN {X 0,Y 467.006,Z 767.116,A -85,B 0,C 180,E1 -7657.567,E2 -7657.567} C_VEL
LIN {X 0,Y 467.208,Z 760.147,A -85,B 0,C 180,E1 -7658.87,E2 -7658.87} C_VEL
LIN {X 0,Y 467.471,Z 751.452,A -85,B 0,C 180,E1 -7660.175,E2 -7660.175} C_VEL
LIN {X 0,Y 467.939,Z 741.511,A -85,B 0,C 180,E1 -7661.37,E2 -7661.37} C_VEL
LIN {X 0,Y 468.46,Z 729.493,A -85,B 0,C 180,E1 -7662.541,E2 -7662.541} C_VEL
LIN {X 0,Y 468.941,Z 718.077,A -85,B 0,C 180,E1 -7663.433,E2 -7663.433} C_VEL
LIN {X 0,Y 469.466,Z 705.63,A -85,B 0,C 180,E1 -7664.191,E2 -7664.191} C_VEL
LIN {X 0,Y 469.786,Z 693.86,A -85,B 0,C 180,E1 -7664.734,E2 -7664.734} C_VEL
LIN {X 0,Y 468.452,Z 682.156,A -85,B 0,C 180,E1 -7665.166,E2 -7665.166} C_VEL
LIN {X 0,Y 467.364,Z 671.036,A -85,B 0,C 180,E1 -7665.454,E2 -7665.454} C_VEL
LIN {X 0,Y 467.685,Z 657.742,A -85,B 0,C 180,E1 -7668.396,E2 -7668.396} C_VEL
LIN {X 0,Y 468.001,Z 643.122,A -85,B 0,C 180,E1 -7671.673,E2 -7671.673} C_VEL
LIN {X 0,Y 468.46,Z 628.119,A -85,B 0,C 180,E1 -7675.076,E2 -7675.076} C_VEL
LIN {X 0,Y 468.811,Z 616.297,A -85,B 0,C 180,E1 -7677.812,E2 -7677.812} C_VEL
LIN {X 0,Y 469.259,Z 604.439,A -85,B 0,C 180,E1 -7680.612,E2 -7680.612} C_VEL
LIN {X 0,Y 469.788,Z 592.027,A -85,B 0,C 180,E1 -7683.609,E2 -7683.609} C_VEL
LIN {X 0,Y 470.214,Z 580.853,A -85,B 0,C 180,E1 -7686.398,E2 -7686.398} C_VEL
LIN {X 0,Y 469.077,Z 573.719,A -85,B 0,C 180,E1 -7688.318,E2 -7688.318} C_VEL
LIN {X 0,Y 467.604,Z 566.241,A -85,B 0,C 180,E1 -7690.474,E2 -7690.474} C_VEL
LIN {X 0,Y 467.561,Z 566.246,A -85,B 0,C 180,E1 -7693.744,E2 -7693.744} C_VEL
LIN {X 0,Y 467.561,Z 566.246,A -85,B 0,C 180,E1 -7696.256,E2 -7696.256} C_VEL
LIN {X 0,Y 467.583,Z 566.243,A -85,B 0,C 180,E1 -7698.723,E2 -7698.723} C_VEL
LIN {X 0,Y 467.57,Z 566.244,A -85,B 0,C 180,E1 -7701.956,E2 -7701.956} C_VEL
LIN {X 0,Y 467.573,Z 566.242,A -85,B 0,C 180,E1 -7705.168,E2 -7705.168} C_VEL
LIN {X 0,Y 467.587,Z 566.243,A -85,B 0,C 180,E1 -7708.26,E2 -7708.26} C_VEL
LIN {X 0,Y 467.581,Z 566.24,A -85,B 0,C 180,E1 -7711.25,E2 -7711.25} C_VEL
LIN {X 0,Y 467.615,Z 566.239,A -85,B 0,C 180,E1 -7714.16,E2 -7714.16} C_VEL
LIN {X 0,Y 467.581,Z 566.241,A -85,B 0,C 180,E1 -7716.996,E2 -7716.996} C_VEL
LIN {X 0,Y 467.627,Z 566.236,A -85,B 0,C 180,E1 -7719.777,E2 -7719.777} C_VEL
LIN {X 0,Y 467.613,Z 566.24,A -85,B 0,C 180,E1 -7722.507,E2 -7722.507} C_VEL
LIN {X 0,Y 467.61,Z 566.237,A -85,B 0,C 180,E1 -7725.196,E2 -7725.196} C_VEL
LIN {X 0,Y 467.66,Z 566.232,A -85,B 0,C 180,E1 -7727.854,E2 -7727.854} C_VEL
LIN {X 0,Y 467.686,Z 566.227,A -85,B 0,C 180,E1 -7731.357,E2 -7731.357} C_VEL
LIN {X 0,Y 467.748,Z 566.221,A -85,B 0,C 180,E1 -7733.962,E2 -7733.962} C_VEL
LIN {X 0,Y 467.862,Z 566.206,A -85,B 0,C 180,E1 -7737.417,E2 -7737.417} C_VEL
LIN {X 0,Y 467.886,Z 566.205,A -85,B 0,C 180,E1 -7740,E2 -7740} C_VEL
LIN {X 0,Y 467.862,Z 566.208,A -85,B 0,C 180,E1 -7742.583,E2 -7742.583} C_VEL
LIN {X 0,Y 467.747,Z 566.223,A -85,B 0,C 180,E1 -7746.037,E2 -7746.037} C_VEL
LIN {X 0,Y 467.684,Z 566.23,A -85,B 0,C 180,E1 -7748.642,E2 -7748.642} C_VEL
LIN {X 0,Y 467.659,Z 566.233,A -85,B 0,C 180,E1 -7752.145,E2 -7752.145} C_VEL
LIN {X 0,Y 467.642,Z 566.234,A -85,B 0,C 180,E1 -7755.695,E2 -7755.695} C_VEL
LIN {X 0,Y 467.62,Z 566.238,A -85,B 0,C 180,E1 -7758.764,E2 -7758.764} C_VEL
LIN {X 0,Y 467.583,Z 566.241,A -85,B 0,C 180,E1 -7761.268,E2 -7761.268} C_VEL
LIN {X 0,Y 467.576,Z 566.243,A -85,B 0,C 180,E1 -7763.943,E2 -7763.943} C_VEL
LIN {X 0,Y 467.619,Z 566.239,A -85,B 0,C 180,E1 -7766.8,E2 -7766.8} C_VEL
LIN {X 0,Y 467.556,Z 566.245,A -85,B 0,C 180,E1 -7769.738,E2 -7769.738} C_VEL
LIN {X 0,Y 467.585,Z 566.243,A -85,B 0,C 180,E1 -7772.758,E2 -7772.758} C_VEL
LIN {X 0,Y 467.558,Z 566.244,A -85,B 0,C 180,E1 -7775.889,E2 -7775.889} C_VEL
LIN {X 0,Y 467.584,Z 566.241,A -85,B 0,C 180,E1 -7779.144,E2 -7779.144} C_VEL
LIN {X 0,Y 467.588,Z 566.242,A -85,B 0,C 180,E1 -7782.566,E2 -7782.566} C_VEL
LIN {X 0,Y 467.572,Z 566.243,A -85,B 0,C 180,E1 -7785.053,E2 -7785.053} C_VEL
LIN {X 0,Y 467.59,Z 566.24,A -85,B 0,C 180,E1 -7787.439,E2 -7787.439} C_VEL
LIN {X 0,Y 467.583,Z 566.242,A -85,B 0,C 180,E1 -7790.855,E2 -7790.855} C_VEL
LIN {X 0,Y 467.56,Z 566.246,A -85,B 0,C 180,E1 -7794.26,E2 -7794.26} C_VEL
LIN {X 0,Y 467.583,Z 566.241,A -85,B 0,C 180,E1 -7797.32,E2 -7797.32} C_VEL
LIN {X 0,Y 467.571,Z 566.246,A -85,B 0,C 180,E1 -7800.667,E2 -7800.667} C_VEL
LIN {X 0,Y 467.617,Z 566.237,A -85,B 0,C 180,E1 -7803.199,E2 -7803.199} C_VEL
LIN {X 0,Y 467.593,Z 566.242,A -85,B 0,C 180,E1 -7806.467,E2 -7806.467} C_VEL
LIN {X 0,Y 467.623,Z 566.235,A -85,B 0,C 180,E1 -7809.777,E2 -7809.777} C_VEL
LIN {X 0,Y 467.609,Z 566.241,A -85,B 0,C 180,E1 -7812.506,E2 -7812.506} C_VEL
LIN {X 0,Y 467.597,Z 566.238,A -85,B 0,C 180,E1 -7815.421,E2 -7815.421} C_VEL
LIN {X 0,Y 466.929,Z 566.325,A -85,B 0,C 180,E1 -7816.14,E2 -7816.14} C_VEL
LIN {X 0,Y 464.094,Z 566.675,A -85,B 0,C 180,E1 -7817.309,E2 -7817.309} C_VEL
LIN {X 0,Y 461.7,Z 566.976,A -85,B 0,C 180,E1 -7818.251,E2 -7818.251} C_VEL
LIN {X 0,Y 460.671,Z 567.104,A -85,B 0,C 180,E1 -7818.979,E2 -7818.979} C_VEL
LIN {X 0,Y 460.587,Z 567.112,A -85,B 0,C 180,E1 -7819.226,E2 -7819.226} C_VEL
LIN {X 0,Y 460.719,Z 567.098,A -85,B 0,C 180,E1 -7822.537,E2 -7822.537} C_VEL
LIN {X 0,Y 460.698,Z 567.101,A -85,B 0,C 180,E1 -7824.748,E2 -7824.748} C_VEL
LIN {X 0,Y 460.825,Z 567.086,A -85,B 0,C 180,E1 -7827.377,E2 -7827.377} C_VEL
LIN {X 0,Y 460.805,Z 567.139,A -85,B 0,C 180,E1 -7829.235,E2 -7829.235} C_VEL
LIN {X 0,Y 463.581,Z 577.787,A -85,B 0,C 180,E1 -7829.891,E2 -7829.891} C_VEL
LIN {X 0,Y 463.224,Z 589.21,A -85,B 0,C 180,E1 -7830.651,E2 -7830.651} C_VEL
LIN {X 0,Y 462.696,Z 600.716,A -85,B 0,C 180,E1 -7831.631,E2 -7831.631} C_VEL
LIN {X 0,Y 462.33,Z 609.961,A -85,B 0,C 180,E1 -7832.613,E2 -7832.613} C_VEL
LIN {X 0,Y 461.864,Z 618.456,A -85,B 0,C 180,E1 -7833.707,E2 -7833.707} C_VEL
LIN {X 0,Y 461.473,Z 626.682,A -85,B 0,C 180,E1 -7835.023,E2 -7835.023} C_VEL
LIN {X 0,Y 461.212,Z 632.32,A -85,B 0,C 180,E1 -7836.122,E2 -7836.122} C_VEL
LIN {X 0,Y 460.879,Z 638.43,A -85,B 0,C 180,E1 -7837.612,E2 -7837.612} C_VEL
LIN {X 0,Y 460.595,Z 643.405,A -85,B 0,C 180,E1 -7839.218,E2 -7839.218} C_VEL
LIN {X 0,Y 460.435,Z 646.35,A -85,B 0,C 180,E1 -7840.553,E2 -7840.553} C_VEL
LIN {X 0,Y 460.332,Z 648.711,A -85,B 0,C 180,E1 -7842.286,E2 -7842.286} C_VEL
LIN {X 0,Y 460.29,Z 649.38,A -85,B 0,C 180,E1 -7843.239,E2 -7843.239} C_VEL
LIN {X 0,Y 460.269,Z 649.593,A -85,B 0,C 180,E1 -7844.14,E2 -7844.14} C_VEL
LIN {X 0,Y 460.316,Z 648.808,A -85,B 0,C 180,E1 -7845.874,E2 -7845.874} C_VEL
LIN {X 0,Y 460.391,Z 647.719,A -85,B 0,C 180,E1 -7846.859,E2 -7846.859} C_VEL
LIN {X 0,Y 460.483,Z 646.217,A -85,B 0,C 180,E1 -7847.772,E2 -7847.772} C_VEL
LIN {X 0,Y 460.657,Z 643.69,A -85,B 0,C 180,E1 -7848.934,E2 -7848.934} C_VEL
LIN {X 0,Y 460.939,Z 638.879,A -85,B 0,C 180,E1 -7850.528,E2 -7850.528} C_VEL
LIN {X 0,Y 461.295,Z 633.419,A -85,B 0,C 180,E1 -7851.899,E2 -7851.899} C_VEL
LIN {X 0,Y 461.704,Z 626.306,A -85,B 0,C 180,E1 -7853.313,E2 -7853.313} C_VEL
LIN {X 0,Y 462.153,Z 618.975,A -85,B 0,C 180,E1 -7854.48,E2 -7854.48} C_VEL
LIN {X 0,Y 462.642,Z 609.919,A -85,B 0,C 180,E1 -7855.653,E2 -7855.653} C_VEL
LIN {X 0,Y 463.075,Z 600.416,A -85,B 0,C 180,E1 -7856.658,E2 -7856.658} C_VEL
LIN {X 0,Y 463.523,Z 590.063,A -85,B 0,C 180,E1 -7857.544,E2 -7857.544} C_VEL
LIN {X 0,Y 463.914,Z 579.388,A -85,B 0,C 180,E1 -7858.272,E2 -7858.272} C_VEL
LIN {X 0,Y 463.133,Z 575.41,A -85,B 0,C 180,E1 -7858.538,E2 -7858.538} C_VEL
LIN {X 0,Y 460.573,Z 567.118,A -85,B 0,C 180,E1 -7859.084,E2 -7859.084} C_VEL
LIN {X 0,Y 460.527,Z 567.121,A -85,B 0,C 180,E1 -7862.284,E2 -7862.284} C_VEL
LIN {X 0,Y 460.506,Z 567.124,A -85,B 0,C 180,E1 -7865.445,E2 -7865.445} C_VEL
LIN {X 0,Y 460.559,Z 567.119,A -85,B 0,C 180,E1 -7868.9,E2 -7868.9} C_VEL
LIN {X 0,Y 460.63,Z 567.272,A -85,B 0,C 180,E1 -7869.591,E2 -7869.591} C_VEL
LIN {X 0,Y 461.294,Z 572.625,A -85,B 0,C 180,E1 -7871.71,E2 -7871.71} C_VEL
LIN {X 0,Y 461.184,Z 581.248,A -85,B 0,C 180,E1 -7874.999,E2 -7874.999} C_VEL
LIN {X 0,Y 461.08,Z 588.88,A -85,B 0,C 180,E1 -7877.882,E2 -7877.882} C_VEL
LIN {X 0,Y 460.838,Z 597.171,A -85,B 0,C 180,E1 -7881.055,E2 -7881.055} C_VEL
LIN {X 0,Y 460.723,Z 604.719,A -85,B 0,C 180,E1 -7883.945,E2 -7883.945} C_VEL
LIN {X 0,Y 460.573,Z 612.831,A -85,B 0,C 180,E1 -7887.06,E2 -7887.06} C_VEL
LIN {X 0,Y 460.405,Z 619.855,A -85,B 0,C 180,E1 -7889.753,E2 -7889.753} C_VEL
LIN {X 0,Y 460.256,Z 624.313,A -85,B 0,C 180,E1 -7891.447,E2 -7891.447} C_VEL
LIN {X 0,Y 463.083,Z 638.406,A -85,B 0,C 180,E1 -7891.958,E2 -7891.958} C_VEL
LIN {X 0,Y 463.297,Z 642.625,A -85,B 0,C 180,E1 -7892.126,E2 -7892.126} C_VEL
LIN {X 0,Y 462.856,Z 654.665,A -85,B 0,C 180,E1 -7892.686,E2 -7892.686} C_VEL
LIN {X 0,Y 462.485,Z 665.789,A -85,B 0,C 180,E1 -7893.367,E2 -7893.367} C_VEL
LIN {X 0,Y 461.953,Z 676.355,A -85,B 0,C 180,E1 -7894.184,E2 -7894.184} C_VEL
LIN {X 0,Y 461.461,Z 687.271,A -85,B 0,C 180,E1 -7895.24,E2 -7895.24} C_VEL
LIN {X 0,Y 460.973,Z 696.919,A -85,B 0,C 180,E1 -7896.395,E2 -7896.395} C_VEL
LIN {X 0,Y 460.533,Z 704.91,A -85,B 0,C 180,E1 -7897.573,E2 -7897.573} C_VEL
LIN {X 0,Y 460.199,Z 712.912,A -85,B 0,C 180,E1 -7899.04,E2 -7899.04} C_VEL
LIN {X 0,Y 459.95,Z 718.6,A -85,B 0,C 180,E1 -7900.357,E2 -7900.357} C_VEL
LIN {X 0,Y 459.768,Z 723.368,A -85,B 0,C 180,E1 -7901.784,E2 -7901.784} C_VEL
LIN {X 0,Y 459.629,Z 726.688,A -85,B 0,C 180,E1 -7903.111,E2 -7903.111} C_VEL
LIN {X 0,Y 459.584,Z 729.019,A -85,B 0,C 180,E1 -7904.446,E2 -7904.446} C_VEL
LIN {X 0,Y 459.489,Z 730.433,A -85,B 0,C 180,E1 -7905.835,E2 -7905.835} C_VEL
LIN {X 0,Y 459.496,Z 730.803,A -85,B 0,C 180,E1 -7906.737,E2 -7906.737} C_VEL
LIN {X 0,Y 459.587,Z 730.544,A -85,B 0,C 180,E1 -7908.143,E2 -7908.143} C_VEL
LIN {X 0,Y 459.597,Z 729.411,A -85,B 0,C 180,E1 -7909.427,E2 -7909.427} C_VEL
LIN {X 0,Y 459.596,Z 728.126,A -85,B 0,C 180,E1 -7910.317,E2 -7910.317} C_VEL
LIN {X 0,Y 459.768,Z 725.355,A -85,B 0,C 180,E1 -7911.651,E2 -7911.651} C_VEL
LIN {X 0,Y 459.907,Z 721.564,A -85,B 0,C 180,E1 -7912.978,E2 -7912.978} C_VEL
LIN {X 0,Y 460.063,Z 716.652,A -85,B 0,C 180,E1 -7914.302,E2 -7914.302} C_VEL
LIN {X 0,Y 460.319,Z 710.44,A -85,B 0,C 180,E1 -7915.622,E2 -7915.622} C_VEL
LIN {X 0,Y 460.651,Z 702.708,A -85,B 0,C 180,E1 -7916.939,E2 -7916.939} C_VEL
LIN {X 0,Y 461.103,Z 694.824,A -85,B 0,C 180,E1 -7918.035,E2 -7918.035} C_VEL
LIN {X 0,Y 461.631,Z 685.255,A -85,B 0,C 180,E1 -7919.128,E2 -7919.128} C_VEL
LIN {X 0,Y 462.126,Z 674.56,A -85,B 0,C 180,E1 -7920.109,E2 -7920.109} C_VEL
LIN {X 0,Y 462.677,Z 662.612,A -85,B 0,C 180,E1 -7920.979,E2 -7920.979} C_VEL
LIN {X 0,Y 463.135,Z 650.967,A -85,B 0,C 180,E1 -7921.631,E2 -7921.631} C_VEL
LIN {X 0,Y 463.33,Z 639.468,A -85,B 0,C 180,E1 -7922.119,E2 -7922.119} C_VEL
LIN {X 0,Y 461.011,Z 628.336,A -85,B 0,C 180,E1 -7922.546,E2 -7922.546} C_VEL
LIN {X 0,Y 460.264,Z 625.43,A -85,B 0,C 180,E1 -7922.681,E2 -7922.681} C_VEL
LIN {X 0,Y 460.6,Z 619.75,A -85,B 0,C 180,E1 -7924.814,E2 -7924.814} C_VEL
LIN {X 0,Y 460.772,Z 610.407,A -85,B 0,C 180,E1 -7928.332,E2 -7928.332} C_VEL
LIN {X 0,Y 460.887,Z 602.036,A -85,B 0,C 180,E1 -7931.434,E2 -7931.434} C_VEL
LIN {X 0,Y 460.996,Z 595.869,A -85,B 0,C 180,E1 -7933.669,E2 -7933.669} C_VEL
LIN {X 0,Y 461.029,Z 588.737,A -85,B 0,C 180,E1 -7936.186,E2 -7936.186} C_VEL
LIN {X 0,Y 461.114,Z 580.258,A -85,B 0,C 180,E1 -7939.101,E2 -7939.101} C_VEL
LIN {X 0,Y 461.084,Z 571.689,A -85,B 0,C 180,E1 -7941.928,E2 -7941.928} C_VEL
LIN {X 0,Y 460.564,Z 567.12,A -85,B 0,C 180,E1 -7943.493,E2 -7943.493} C_VEL
LIN {X 0,Y 460.562,Z 567.12,A -85,B 0,C 180,E1 -7946.266,E2 -7946.266} C_VEL
LIN {X 0,Y 460.542,Z 567.121,A -85,B 0,C 180,E1 -7949.231,E2 -7949.231} C_VEL
LIN {X 0,Y 460.527,Z 567.123,A -85,B 0,C 180,E1 -7952.285,E2 -7952.285} C_VEL
LIN {X 0,Y 460.509,Z 567.124,A -85,B 0,C 180,E1 -7955.446,E2 -7955.446} C_VEL
LIN {X 0,Y 460.561,Z 567.117,A -85,B 0,C 180,E1 -7958.902,E2 -7958.902} C_VEL
LIN {X 0,Y 460.544,Z 567.115,A -85,B 0,C 180,E1 -7962.179,E2 -7962.179} C_VEL
LIN {X 0,Y 460.518,Z 567.123,A -85,B 0,C 180,E1 -7965.413,E2 -7965.413} C_VEL
LIN {X 0,Y 460.542,Z 567.118,A -85,B 0,C 180,E1 -7968.397,E2 -7968.397} C_VEL
LIN {X 0,Y 460.609,Z 567.328,A -85,B 0,C 180,E1 -7968.878,E2 -7968.878} C_VEL
LIN {X 0,Y 462.28,Z 575.639,A -85,B 0,C 180,E1 -7971.442,E2 -7971.442} C_VEL
LIN {X 0,Y 463.449,Z 582.657,A -85,B 0,C 180,E1 -7973.488,E2 -7973.488} C_VEL
LIN {X 0,Y 462.903,Z 593.249,A -85,B 0,C 180,E1 -7976.285,E2 -7976.285} C_VEL
LIN {X 0,Y 462.249,Z 606.569,A -85,B 0,C 180,E1 -7979.635,E2 -7979.635} C_VEL
LIN {X 0,Y 461.709,Z 619.693,A -85,B 0,C 180,E1 -7982.83,E2 -7982.83} C_VEL
LIN {X 0,Y 461.229,Z 633.569,A -85,B 0,C 180,E1 -7986.1,E2 -7986.1} C_VEL
LIN {X 0,Y 460.752,Z 648.159,A -85,B 0,C 180,E1 -7989.463,E2 -7989.463} C_VEL
LIN {X 0,Y 460.487,Z 661.39,A -85,B 0,C 180,E1 -7992.458,E2 -7992.458} C_VEL
LIN {X 0,Y 460.295,Z 669.833,A -85,B 0,C 180,E1 -7994.309,E2 -7994.309} C_VEL
LIN {X 0,Y 461.637,Z 683.447,A -85,B 0,C 180,E1 -7994.679,E2 -7994.679} C_VEL
LIN {X 0,Y 462.774,Z 693.953,A -85,B 0,C 180,E1 -7995.096,E2 -7995.096} C_VEL
LIN {X 0,Y 462.478,Z 705.382,A -85,B 0,C 180,E1 -7995.648,E2 -7995.648} C_VEL
LIN {X 0,Y 461.924,Z 716.799,A -85,B 0,C 180,E1 -7996.361,E2 -7996.361} C_VEL
LIN {X 0,Y 461.389,Z 728.311,A -85,B 0,C 180,E1 -7997.275,E2 -7997.275} C_VEL
LIN {X 0,Y 460.818,Z 741.409,A -85,B 0,C 180,E1 -7998.565,E2 -7998.565} C_VEL
LIN {X 0,Y 460.434,Z 750.444,A -85,B 0,C 180,E1 -7999.669,E2 -7999.669} C_VEL
LIN {X 0,Y 460.145,Z 759.275,A -85,B 0,C 180,E1 -8000.994,E2 -8000.994} C_VEL
LIN {X 0,Y 459.937,Z 766.309,A -85,B 0,C 180,E1 -8002.317,E2 -8002.317} C_VEL
LIN {X 0,Y 459.806,Z 772.768,A -85,B 0,C 180,E1 -8003.859,E2 -8003.859} C_VEL
LIN {X 0,Y 459.741,Z 776.962,A -85,B 0,C 180,E1 -8005.178,E2 -8005.178} C_VEL
LIN {X 0,Y 459.766,Z 780.056,A -85,B 0,C 180,E1 -8006.495,E2 -8006.495} C_VEL
LIN {X 0,Y 459.717,Z 781.551,A -85,B 0,C 180,E1 -8007.372,E2 -8007.372} C_VEL
LIN {X 0,Y 459.718,Z 782.608,A -85,B 0,C 180,E1 -8008.249,E2 -8008.249} C_VEL
LIN {X 0,Y 459.673,Z 783.257,A -85,B 0,C 180,E1 -8009.125,E2 -8009.125} C_VEL
LIN {X 0,Y 459.662,Z 783.496,A -85,B 0,C 180,E1 -8010.001,E2 -8010.001} C_VEL
LIN {X 0,Y 459.672,Z 783.292,A -85,B 0,C 180,E1 -8010.877,E2 -8010.877} C_VEL
LIN {X 0,Y 459.72,Z 782.675,A -85,B 0,C 180,E1 -8011.753,E2 -8011.753} C_VEL
LIN {X 0,Y 459.719,Z 781.651,A -85,B 0,C 180,E1 -8012.629,E2 -8012.629} C_VEL
LIN {X 0,Y 459.746,Z 780.192,A -85,B 0,C 180,E1 -8013.506,E2 -8013.506} C_VEL
LIN {X 0,Y 459.731,Z 777.171,A -85,B 0,C 180,E1 -8014.824,E2 -8014.824} C_VEL
LIN {X 0,Y 459.808,Z 773.043,A -85,B 0,C 180,E1 -8016.143,E2 -8016.143} C_VEL
LIN {X 0,Y 459.927,Z 766.693,A -85,B 0,C 180,E1 -8017.685,E2 -8017.685} C_VEL
LIN {X 0,Y 460.145,Z 759.737,A -85,B 0,C 180,E1 -8019.008,E2 -8019.008} C_VEL
LIN {X 0,Y 460.435,Z 751.007,A -85,B 0,C 180,E1 -8020.333,E2 -8020.333} C_VEL
LIN {X 0,Y 460.931,Z 741.065,A -85,B 0,C 180,E1 -8021.545,E2 -8021.545} C_VEL
LIN {X 0,Y 461.404,Z 730.49,A -85,B 0,C 180,E1 -8022.576,E2 -8022.576} C_VEL
LIN {X 0,Y 461.982,Z 717.046,A -85,B 0,C 180,E1 -8023.639,E2 -8023.639} C_VEL
LIN {X 0,Y 462.554,Z 704.565,A -85,B 0,C 180,E1 -8024.407,E2 -8024.407} C_VEL
LIN {X 0,Y 462.766,Z 694.056,A -85,B 0,C 180,E1 -8024.906,E2 -8024.906} C_VEL
LIN {X 0,Y 461.559,Z 683.352,A -85,B 0,C 180,E1 -8025.325,E2 -8025.325} C_VEL
LIN {X 0,Y 460.297,Z 670.018,A -85,B 0,C 180,E1 -8025.693,E2 -8025.693} C_VEL
LIN {X 0,Y 460.649,Z 655.718,A -85,B 0,C 180,E1 -8028.929,E2 -8028.929} C_VEL
LIN {X 0,Y 460.983,Z 641.511,A -85,B 0,C 180,E1 -8032.169,E2 -8032.169} C_VEL
LIN {X 0,Y 461.416,Z 628.211,A -85,B 0,C 180,E1 -8035.245,E2 -8035.245} C_VEL
LIN {X 0,Y 461.826,Z 615.89,A -85,B 0,C 180,E1 -8038.149,E2 -8038.149} C_VEL
LIN {X 0,Y 462.273,Z 604.56,A -85,B 0,C 180,E1 -8040.872,E2 -8040.872} C_VEL
LIN {X 0,Y 462.819,Z 593.021,A -85,B 0,C 180,E1 -8043.711,E2 -8043.711} C_VEL
LIN {X 0,Y 463.264,Z 582.07,A -85,B 0,C 180,E1 -8046.482,E2 -8046.482} C_VEL
LIN {X 0,Y 461.966,Z 574.366,A -85,B 0,C 180,E1 -8048.591,E2 -8048.591} C_VEL
LIN {X 0,Y 460.55,Z 567.12,A -85,B 0,C 180,E1 -8050.713,E2 -8050.713} C_VEL
LIN {X 0,Y 460.516,Z 567.124,A -85,B 0,C 180,E1 -8054.17,E2 -8054.17} C_VEL
LIN {X 0,Y 460.518,Z 567.123,A -85,B 0,C 180,E1 -8057.1,E2 -8057.1} C_VEL
LIN {X 0,Y 460.562,Z 567.118,A -85,B 0,C 180,E1 -8060.14,E2 -8060.14} C_VEL
LIN {X 0,Y 460.484,Z 567.124,A -85,B 0,C 180,E1 -8063.471,E2 -8063.471} C_VEL
LIN {X 0,Y 460.534,Z 567.12,A -85,B 0,C 180,E1 -8066.675,E2 -8066.675} C_VEL
LIN {X 0,Y 460.515,Z 567.123,A -85,B 0,C 180,E1 -8069.76,E2 -8069.76} C_VEL
LIN {X 0,Y 460.578,Z 567.116,A -85,B 0,C 180,E1 -8072.756,E2 -8072.756} C_VEL
LIN {X 0,Y 460.546,Z 567.118,A -85,B 0,C 180,E1 -8075.668,E2 -8075.668} C_VEL
LIN {X 0,Y 460.526,Z 567.122,A -85,B 0,C 180,E1 -8078.578,E2 -8078.578} C_VEL
LIN {X 0,Y 460.595,Z 567.112,A -85,B 0,C 180,E1 -8081.311,E2 -8081.311} C_VEL
LIN {X 0,Y 460.608,Z 567.112,A -85,B 0,C 180,E1 -8084.059,E2 -8084.059} C_VEL
LIN {X 0,Y 460.613,Z 567.11,A -85,B 0,C 180,E1 -8087.666,E2 -8087.666} C_VEL
LIN {X 0,Y 460.633,Z 567.106,A -85,B 0,C 180,E1 -8091.224,E2 -8091.224} C_VEL
LIN {X 0,Y 460.714,Z 567.097,A -85,B 0,C 180,E1 -8093.87,E2 -8093.87} C_VEL
LIN {X 0,Y 460.802,Z 567.085,A -85,B 0,C 180,E1 -8097.377,E2 -8097.377} C_VEL
LIN {X 0,Y 460.857,Z 567.08,A -85,B 0,C 180,E1 -8100,E2 -8100} C_VEL
LIN {X 0,Y 460.803,Z 567.087,A -85,B 0,C 180,E1 -8102.622,E2 -8102.622} C_VEL
LIN {X 0,Y 460.713,Z 567.099,A -85,B 0,C 180,E1 -8106.13,E2 -8106.13} C_VEL
LIN {X 0,Y 460.632,Z 567.108,A -85,B 0,C 180,E1 -8108.776,E2 -8108.776} C_VEL
LIN {X 0,Y 460.617,Z 567.111,A -85,B 0,C 180,E1 -8112.444,E2 -8112.444} C_VEL
LIN {X 0,Y 460.603,Z 567.111,A -85,B 0,C 180,E1 -8115.997,E2 -8115.997} C_VEL
LIN {X 0,Y 460.573,Z 567.115,A -85,B 0,C 180,E1 -8118.901,E2 -8118.901} C_VEL
LIN {X 0,Y 460.519,Z 567.12,A -85,B 0,C 180,E1 -8121.485,E2 -8121.485} C_VEL
LIN {X 0,Y 460.545,Z 567.12,A -85,B 0,C 180,E1 -8124.332,E2 -8124.332} C_VEL
LIN {X 0,Y 460.575,Z 567.113,A -85,B 0,C 180,E1 -8127.243,E2 -8127.243} C_VEL
LIN {X 0,Y 460.512,Z 567.124,A -85,B 0,C 180,E1 -8130.239,E2 -8130.239} C_VEL
LIN {X 0,Y 460.531,Z 567.119,A -85,B 0,C 180,E1 -8133.324,E2 -8133.324} C_VEL
LIN {X 0,Y 460.481,Z 567.128,A -85,B 0,C 180,E1 -8136.529,E2 -8136.529} C_VEL
LIN {X 0,Y 460.546,Z 567.118,A -85,B 0,C 180,E1 -8138.897,E2 -8138.897} C_VEL
LIN {X 0,Y 460.525,Z 567.123,A -85,B 0,C 180,E1 -8142.181,E2 -8142.181} C_VEL
LIN {X 0,Y 460.521,Z 567.121,A -85,B 0,C 180,E1 -8145.411,E2 -8145.411} C_VEL
LIN {X 0,Y 460.536,Z 567.121,A -85,B 0,C 180,E1 -8148.396,E2 -8148.396} C_VEL
LIN {X 0,Y 460.527,Z 567.12,A -85,B 0,C 180,E1 -8151.266,E2 -8151.266} C_VEL
LIN {X 0,Y 460.511,Z 567.124,A -85,B 0,C 180,E1 -8154.554,E2 -8154.554} C_VEL
LIN {X 0,Y 460.533,Z 567.119,A -85,B 0,C 180,E1 -8157.715,E2 -8157.715} C_VEL
LIN {X 0,Y 460.541,Z 567.121,A -85,B 0,C 180,E1 -8160.768,E2 -8160.768} C_VEL
LIN {X 0,Y 460.563,Z 567.115,A -85,B 0,C 180,E1 -8163.734,E2 -8163.734} C_VEL
LIN {X 0,Y 460.546,Z 567.121,A -85,B 0,C 180,E1 -8166.623,E2 -8166.623} C_VEL
LIN {X 0,Y 460.552,Z 567.116,A -85,B 0,C 180,E1 -8169.452,E2 -8169.452} C_VEL
LIN {X 0,Y 460.559,Z 567.117,A -85,B 0,C 180,E1 -8172.229,E2 -8172.229} C_VEL
LIN {X 0,Y 460.565,Z 567.116,A -85,B 0,C 180,E1 -8174.964,E2 -8174.964} C_VEL
LIN {X 0,Y 460.629,Z 567.106,A -85,B 0,C 180,E1 -8177.666,E2 -8177.666} C_VEL
LIN {X 0,Y 460.587,Z 567.112,A -85,B 0,C 180,E1 -8179.226,E2 -8179.226} C_VEL
LIN {X 0,Y 459.925,Z 567.196,A -85,B 0,C 180,E1 -8179.956,E2 -8179.956} C_VEL
LIN {X 0,Y 457.103,Z 567.552,A -85,B 0,C 180,E1 -8181.142,E2 -8181.142} C_VEL
LIN {X 0,Y 454.725,Z 567.848,A -85,B 0,C 180,E1 -8182.099,E2 -8182.099} C_VEL
LIN {X 0,Y 453.713,Z 567.971,A -85,B 0,C 180,E1 -8182.838,E2 -8182.838} C_VEL
LIN {X 0,Y 453.636,Z 567.979,A -85,B 0,C 180,E1 -8183.088,E2 -8183.088} C_VEL
LIN {X 0,Y 453.671,Z 567.976,A -85,B 0,C 180,E1 -8184.666,E2 -8184.666} C_VEL
LIN {X 0,Y 453.765,Z 567.965,A -85,B 0,C 180,E1 -8187.336,E2 -8187.336} C_VEL
LIN {X 0,Y 453.71,Z 567.972,A -85,B 0,C 180,E1 -8189.001,E2 -8189.001} C_VEL
LIN {X 0,Y 456.616,Z 578.378,A -85,B 0,C 180,E1 -8189.668,E2 -8189.668} C_VEL
LIN {X 0,Y 456.369,Z 589.863,A -85,B 0,C 180,E1 -8190.44,E2 -8190.44} C_VEL
LIN {X 0,Y 455.827,Z 601.428,A -85,B 0,C 180,E1 -8191.435,E2 -8191.435} C_VEL
LIN {X 0,Y 455.444,Z 610.719,A -85,B 0,C 180,E1 -8192.431,E2 -8192.431} C_VEL
LIN {X 0,Y 454.949,Z 619.257,A -85,B 0,C 180,E1 -8193.542,E2 -8193.542} C_VEL
LIN {X 0,Y 454.531,Z 627.531,A -85,B 0,C 180,E1 -8194.878,E2 -8194.878} C_VEL
LIN {X 0,Y 454.174,Z 634.196,A -85,B 0,C 180,E1 -8196.218,E2 -8196.218} C_VEL
LIN {X 0,Y 453.859,Z 639.95,A -85,B 0,C 180,E1 -8197.679,E2 -8197.679} C_VEL
LIN {X 0,Y 453.637,Z 643.719,A -85,B 0,C 180,E1 -8198.912,E2 -8198.912} C_VEL
LIN {X 0,Y 453.483,Z 645.95,A -85,B 0,C 180,E1 -8199.815,E2 -8199.815} C_VEL
LIN {X 0,Y 453.393,Z 647.692,A -85,B 0,C 180,E1 -8200.719,E2 -8200.719} C_VEL
LIN {X 0,Y 453.311,Z 649.949,A -85,B 0,C 180,E1 -8202.535,E2 -8202.535} C_VEL
LIN {X 0,Y 453.254,Z 650.482,A -85,B 0,C 180,E1 -8203.448,E2 -8203.448} C_VEL
LIN {X 0,Y 453.273,Z 650.278,A -85,B 0,C 180,E1 -8205.282,E2 -8205.282} C_VEL
LIN {X 0,Y 453.327,Z 649.586,A -85,B 0,C 180,E1 -8206.203,E2 -8206.203} C_VEL
LIN {X 0,Y 453.412,Z 648.43,A -85,B 0,C 180,E1 -8207.127,E2 -8207.127} C_VEL
LIN {X 0,Y 453.592,Z 645.886,A -85,B 0,C 180,E1 -8208.519,E2 -8208.519} C_VEL
LIN {X 0,Y 453.84,Z 642.258,A -85,B 0,C 180,E1 -8209.918,E2 -8209.918} C_VEL
LIN {X 0,Y 454.174,Z 637.416,A -85,B 0,C 180,E1 -8211.323,E2 -8211.323} C_VEL
LIN {X 0,Y 454.554,Z 631.19,A -85,B 0,C 180,E1 -8212.738,E2 -8212.738} C_VEL
LIN {X 0,Y 455.014,Z 624.113,A -85,B 0,C 180,E1 -8214.025,E2 -8214.025} C_VEL
LIN {X 0,Y 455.468,Z 616.844,A -85,B 0,C 180,E1 -8215.107,E2 -8215.107} C_VEL
LIN {X 0,Y 455.991,Z 607.024,A -85,B 0,C 180,E1 -8216.301,E2 -8216.301} C_VEL
LIN {X 0,Y 456.532,Z 595.917,A -85,B 0,C 180,E1 -8217.38,E2 -8217.38} C_VEL
LIN {X 0,Y 457.044,Z 584.957,A -85,B 0,C 180,E1 -8218.218,E2 -8218.218} C_VEL
LIN {X 0,Y 457.122,Z 579.933,A -85,B 0,C 180,E1 -8218.545,E2 -8218.545} C_VEL
LIN {X 0,Y 453.51,Z 567.997,A -85,B 0,C 180,E1 -8219.358,E2 -8219.358} C_VEL
LIN {X 0,Y 453.477,Z 568.001,A -85,B 0,C 180,E1 -8222.848,E2 -8222.848} C_VEL
LIN {X 0,Y 453.45,Z 568.003,A -85,B 0,C 180,E1 -8226.082,E2 -8226.082} C_VEL
LIN {X 0,Y 453.58,Z 568.178,A -85,B 0,C 180,E1 -8229.439,E2 -8229.439} C_VEL
LIN {X 0,Y 454.311,Z 573.934,A -85,B 0,C 180,E1 -8231.696,E2 -8231.696} C_VEL
LIN {X 0,Y 454.194,Z 581.48,A -85,B 0,C 180,E1 -8234.62,E2 -8234.62} C_VEL
LIN {X 0,Y 454.099,Z 589.224,A -85,B 0,C 180,E1 -8237.576,E2 -8237.576} C_VEL
LIN {X 0,Y 453.859,Z 597.435,A -85,B 0,C 180,E1 -8240.735,E2 -8240.735} C_VEL
LIN {X 0,Y 453.687,Z 605.74,A -85,B 0,C 180,E1 -8243.939,E2 -8243.939} C_VEL
LIN {X 0,Y 453.582,Z 613.135,A -85,B 0,C 180,E1 -8246.791,E2 -8246.791} C_VEL
LIN {X 0,Y 453.317,Z 622.14,A -85,B 0,C 180,E1 -8250.257,E2 -8250.257} C_VEL
LIN {X 0,Y 453.26,Z 624.823,A -85,B 0,C 180,E1 -8251.23,E2 -8251.23} C_VEL
LIN {X 0,Y 456,Z 638.167,A -85,B 0,C 180,E1 -8251.71,E2 -8251.71} C_VEL
LIN {X 0,Y 456.472,Z 641.532,A -85,B 0,C 180,E1 -8251.852,E2 -8251.852} C_VEL
LIN {X 0,Y 455.99,Z 654.64,A -85,B 0,C 180,E1 -8252.46,E2 -8252.46} C_VEL
LIN {X 0,Y 455.568,Z 666.222,A -85,B 0,C 180,E1 -8253.177,E2 -8253.177} C_VEL
LIN {X 0,Y 455.02,Z 677.028,A -85,B 0,C 180,E1 -8254.03,E2 -8254.03} C_VEL
LIN {X 0,Y 454.494,Z 687.682,A -85,B 0,C 180,E1 -8255.079,E2 -8255.079} C_VEL
LIN {X 0,Y 453.98,Z 697.43,A -85,B 0,C 180,E1 -8256.266,E2 -8256.266} C_VEL
LIN {X 0,Y 453.509,Z 705.315,A -85,B 0,C 180,E1 -8257.447,E2 -8257.447} C_VEL
LIN {X 0,Y 453.206,Z 712.602,A -85,B 0,C 180,E1 -8258.791,E2 -8258.791} C_VEL
LIN {X 0,Y 452.922,Z 718.083,A -85,B 0,C 180,E1 -8260.04,E2 -8260.04} C_VEL
LIN {X 0,Y 452.716,Z 723.351,A -85,B 0,C 180,E1 -8261.568,E2 -8261.568} C_VEL
LIN {X 0,Y 452.583,Z 726.625,A -85,B 0,C 180,E1 -8262.84,E2 -8262.84} C_VEL
LIN {X 0,Y 452.497,Z 729.339,A -85,B 0,C 180,E1 -8264.352,E2 -8264.352} C_VEL
LIN {X 0,Y 452.427,Z 730.704,A -85,B 0,C 180,E1 -8265.609,E2 -8265.609} C_VEL
LIN {X 0,Y 452.4,Z 731.167,A -85,B 0,C 180,E1 -8266.525,E2 -8266.525} C_VEL
LIN {X 0,Y 452.513,Z 730.998,A -85,B 0,C 180,E1 -8268.079,E2 -8268.079} C_VEL
LIN {X 0,Y 452.533,Z 730.076,A -85,B 0,C 180,E1 -8269.26,E2 -8269.26} C_VEL
LIN {X 0,Y 452.507,Z 728.867,A -85,B 0,C 180,E1 -8270.163,E2 -8270.163} C_VEL
LIN {X 0,Y 452.671,Z 726.249,A -85,B 0,C 180,E1 -8271.519,E2 -8271.519} C_VEL
LIN {X 0,Y 452.838,Z 722.611,A -85,B 0,C 180,E1 -8272.868,E2 -8272.868} C_VEL
LIN {X 0,Y 452.985,Z 717.868,A -85,B 0,C 180,E1 -8274.212,E2 -8274.212} C_VEL
LIN {X 0,Y 453.26,Z 711.87,A -85,B 0,C 180,E1 -8275.554,E2 -8275.554} C_VEL
LIN {X 0,Y 453.597,Z 704.402,A -85,B 0,C 180,E1 -8276.892,E2 -8276.892} C_VEL
LIN {X 0,Y 454.153,Z 695.049,A -85,B 0,C 180,E1 -8278.227,E2 -8278.227} C_VEL
LIN {X 0,Y 454.718,Z 685.45,A -85,B 0,C 180,E1 -8279.336,E2 -8279.336} C_VEL
LIN {X 0,Y 455.255,Z 674.732,A -85,B 0,C 180,E1 -8280.332,E2 -8280.332} C_VEL
LIN {X 0,Y 455.835,Z 662.78,A -85,B 0,C 180,E1 -8281.215,E2 -8281.215} C_VEL
LIN {X 0,Y 456.327,Z 651.081,A -85,B 0,C 180,E1 -8281.876,E2 -8281.876} C_VEL
LIN {X 0,Y 456.455,Z 639.991,A -85,B 0,C 180,E1 -8282.358,E2 -8282.358} C_VEL
LIN {X 0,Y 454.207,Z 629.731,A -85,B 0,C 180,E1 -8282.772,E2 -8282.772} C_VEL
LIN {X 0,Y 453.311,Z 625.926,A -85,B 0,C 180,E1 -8282.916,E2 -8282.916} C_VEL
LIN {X 0,Y 453.604,Z 619.556,A -85,B 0,C 180,E1 -8285.334,E2 -8285.334} C_VEL
LIN {X 0,Y 453.777,Z 610.063,A -85,B 0,C 180,E1 -8288.91,E2 -8288.91} C_VEL
LIN {X 0,Y 453.976,Z 601.687,A -85,B 0,C 180,E1 -8292.064,E2 -8292.064} C_VEL
LIN {X 0,Y 454.084,Z 592.791,A -85,B 0,C 180,E1 -8295.255,E2 -8295.255} C_VEL
LIN {X 0,Y 454.098,Z 583.496,A -85,B 0,C 180,E1 -8298.499,E2 -8298.499} C_VEL
LIN {X 0,Y 454.152,Z 576.572,A -85,B 0,C 180,E1 -8300.85,E2 -8300.85} C_VEL
LIN {X 0,Y 453.983,Z 570.822,A -85,B 0,C 180,E1 -8302.769,E2 -8302.769} C_VEL
LIN {X 0,Y 453.497,Z 568.001,A -85,B 0,C 180,E1 -8303.762,E2 -8303.762} C_VEL
LIN {X 0,Y 453.507,Z 567.998,A -85,B 0,C 180,E1 -8306.706,E2 -8306.706} C_VEL
LIN {X 0,Y 453.483,Z 568,A -85,B 0,C 180,E1 -8309.79,E2 -8309.79} C_VEL
LIN {X 0,Y 453.485,Z 568.001,A -85,B 0,C 180,E1 -8313.19,E2 -8313.19} C_VEL
LIN {X 0,Y 453.452,Z 568.005,A -85,B 0,C 180,E1 -8316.301,E2 -8316.301} C_VEL
LIN {X 0,Y 453.527,Z 567.995,A -85,B 0,C 180,E1 -8319.446,E2 -8319.446} C_VEL
LIN {X 0,Y 453.488,Z 567.998,A -85,B 0,C 180,E1 -8322.992,E2 -8322.992} C_VEL
LIN {X 0,Y 453.473,Z 568.001,A -85,B 0,C 180,E1 -8325.781,E2 -8325.781} C_VEL
LIN {X 0,Y 453.505,Z 568,A -85,B 0,C 180,E1 -8328.449,E2 -8328.449} C_VEL
LIN {X 0,Y 455.006,Z 575.096,A -85,B 0,C 180,E1 -8330.709,E2 -8330.709} C_VEL
LIN {X 0,Y 456.479,Z 583.334,A -85,B 0,C 180,E1 -8333.188,E2 -8333.188} C_VEL
LIN {X 0,Y 456.197,Z 590.908,A -85,B 0,C 180,E1 -8335.251,E2 -8335.251} C_VEL
LIN {X 0,Y 455.42,Z 603.844,A -85,B 0,C 180,E1 -8338.614,E2 -8338.614} C_VEL
LIN {X 0,Y 454.87,Z 616.278,A -85,B 0,C 180,E1 -8341.725,E2 -8341.725} C_VEL
LIN {X 0,Y 454.273,Z 630.043,A -85,B 0,C 180,E1 -8345.067,E2 -8345.067} C_VEL
LIN {X 0,Y 453.884,Z 642.205,A -85,B 0,C 180,E1 -8347.946,E2 -8347.946} C_VEL
LIN {X 0,Y 453.541,Z 656.372,A -85,B 0,C 180,E1 -8351.245,E2 -8351.245} C_VEL
LIN {X 0,Y 453.248,Z 668.641,A -85,B 0,C 180,E1 -8354.043,E2 -8354.043} C_VEL
LIN {X 0,Y 454.646,Z 682.999,A -85,B 0,C 180,E1 -8354.447,E2 -8354.447} C_VEL
LIN {X 0,Y 455.595,Z 693.015,A -85,B 0,C 180,E1 -8354.855,E2 -8354.855} C_VEL
LIN {X 0,Y 455.917,Z 696.865,A -85,B 0,C 180,E1 -8355.038,E2 -8355.038} C_VEL
LIN {X 0,Y 455.407,Z 707.348,A -85,B 0,C 180,E1 -8355.592,E2 -8355.592} C_VEL
LIN {X 0,Y 454.817,Z 718.817,A -85,B 0,C 180,E1 -8356.371,E2 -8356.371} C_VEL
LIN {X 0,Y 454.291,Z 732.107,A -85,B 0,C 180,E1 -8357.493,E2 -8357.493} C_VEL
LIN {X 0,Y 453.726,Z 742.871,A -85,B 0,C 180,E1 -8358.611,E2 -8358.611} C_VEL
LIN {X 0,Y 453.326,Z 751.598,A -85,B 0,C 180,E1 -8359.731,E2 -8359.731} C_VEL
LIN {X 0,Y 453.051,Z 760.073,A -85,B 0,C 180,E1 -8361.077,E2 -8361.077} C_VEL
LIN {X 0,Y 452.842,Z 766.894,A -85,B 0,C 180,E1 -8362.42,E2 -8362.42} C_VEL
LIN {X 0,Y 452.718,Z 772.324,A -85,B 0,C 180,E1 -8363.762,E2 -8363.762} C_VEL
LIN {X 0,Y 452.668,Z 776.527,A -85,B 0,C 180,E1 -8365.102,E2 -8365.102} C_VEL
LIN {X 0,Y 452.677,Z 779.632,A -85,B 0,C 180,E1 -8366.44,E2 -8366.44} C_VEL
LIN {X 0,Y 452.637,Z 781.13,A -85,B 0,C 180,E1 -8367.331,E2 -8367.331} C_VEL
LIN {X 0,Y 452.652,Z 782.191,A -85,B 0,C 180,E1 -8368.221,E2 -8368.221} C_VEL
LIN {X 0,Y 452.601,Z 782.845,A -85,B 0,C 180,E1 -8369.111,E2 -8369.111} C_VEL
LIN {X 0,Y 452.589,Z 783.092,A -85,B 0,C 180,E1 -8370.001,E2 -8370.001} C_VEL
LIN {X 0,Y 452.601,Z 782.885,A -85,B 0,C 180,E1 -8370.891,E2 -8370.891} C_VEL
LIN {X 0,Y 452.654,Z 782.275,A -85,B 0,C 180,E1 -8371.78,E2 -8371.78} C_VEL
LIN {X 0,Y 452.638,Z 781.259,A -85,B 0,C 180,E1 -8372.671,E2 -8372.671} C_VEL
LIN {X 0,Y 452.658,Z 779.798,A -85,B 0,C 180,E1 -8373.561,E2 -8373.561} C_VEL
LIN {X 0,Y 452.659,Z 776.762,A -85,B 0,C 180,E1 -8374.899,E2 -8374.899} C_VEL
LIN {X 0,Y 452.692,Z 771.728,A -85,B 0,C 180,E1 -8376.486,E2 -8376.486} C_VEL
LIN {X 0,Y 452.893,Z 765.231,A -85,B 0,C 180,E1 -8378.029,E2 -8378.029} C_VEL
LIN {X 0,Y 453.151,Z 757.961,A -85,B 0,C 180,E1 -8379.373,E2 -8379.373} C_VEL
LIN {X 0,Y 453.484,Z 748.906,A -85,B 0,C 180,E1 -8380.719,E2 -8380.719} C_VEL
LIN {X 0,Y 453.911,Z 739.535,A -85,B 0,C 180,E1 -8381.839,E2 -8381.839} C_VEL
LIN {X 0,Y 454.413,Z 729.408,A -85,B 0,C 180,E1 -8382.821,E2 -8382.821} C_VEL
LIN {X 0,Y 454.963,Z 717.613,A -85,B 0,C 180,E1 -8383.74,E2 -8383.74} C_VEL
LIN {X 0,Y 455.573,Z 704.459,A -85,B 0,C 180,E1 -8384.576,E2 -8384.576} C_VEL
LIN {X 0,Y 455.875,Z 695.553,A -85,B 0,C 180,E1 -8385.023,E2 -8385.023} C_VEL
LIN {X 0,Y 454.646,Z 684.013,A -85,B 0,C 180,E1 -8385.507,E2 -8385.507} C_VEL
LIN {X 0,Y 453.364,Z 670.758,A -85,B 0,C 180,E1 -8385.883,E2 -8385.883} C_VEL
LIN {X 0,Y 453.231,Z 669.005,A -85,B 0,C 180,E1 -8385.945,E2 -8385.945} C_VEL
LIN {X 0,Y 453.573,Z 655.46,A -85,B 0,C 180,E1 -8389.059,E2 -8389.059} C_VEL
LIN {X 0,Y 453.914,Z 641.564,A -85,B 0,C 180,E1 -8392.293,E2 -8392.293} C_VEL
LIN {X 0,Y 454.411,Z 627.244,A -85,B 0,C 180,E1 -8395.662,E2 -8395.662} C_VEL
LIN {X 0,Y 454.833,Z 614.939,A -85,B 0,C 180,E1 -8398.621,E2 -8398.621} C_VEL
LIN {X 0,Y 455.296,Z 604.664,A -85,B 0,C 180,E1 -8401.139,E2 -8401.139} C_VEL
LIN {X 0,Y 455.906,Z 592.275,A -85,B 0,C 180,E1 -8404.241,E2 -8404.241} C_VEL
LIN {X 0,Y 456.245,Z 584.329,A -85,B 0,C 180,E1 -8406.295,E2 -8406.295} C_VEL
LIN {X 0,Y 455.799,Z 579.848,A -85,B 0,C 180,E1 -8407.509,E2 -8407.509} C_VEL
LIN {X 0,Y 453.549,Z 568.077,A -85,B 0,C 180,E1 -8410.896,E2 -8410.896} C_VEL
LIN {X 0,Y 453.492,Z 567.999,A -85,B 0,C 180,E1 -8414.529,E2 -8414.529} C_VEL
LIN {X 0,Y 453.484,Z 568,A -85,B 0,C 180,E1 -8418.209,E2 -8418.209} C_VEL
LIN {X 0,Y 453.52,Z 567.994,A -85,B 0,C 180,E1 -8420.79,E2 -8420.79} C_VEL
LIN {X 0,Y 453.462,Z 568.002,A -85,B 0,C 180,E1 -8423.917,E2 -8423.917} C_VEL
LIN {X 0,Y 453.487,Z 567.997,A -85,B 0,C 180,E1 -8427.151,E2 -8427.151} C_VEL
LIN {X 0,Y 453.48,Z 568,A -85,B 0,C 180,E1 -8430.268,E2 -8430.268} C_VEL
LIN {X 0,Y 453.511,Z 567.994,A -85,B 0,C 180,E1 -8433.294,E2 -8433.294} C_VEL
LIN {X 0,Y 453.507,Z 567.996,A -85,B 0,C 180,E1 -8436.239,E2 -8436.239} C_VEL
LIN {X 0,Y 453.487,Z 567.996,A -85,B 0,C 180,E1 -8439.117,E2 -8439.117} C_VEL
LIN {X 0,Y 453.516,Z 567.994,A -85,B 0,C 180,E1 -8441.944,E2 -8441.944} C_VEL
LIN {X 0,Y 453.544,Z 567.992,A -85,B 0,C 180,E1 -8444.726,E2 -8444.726} C_VEL
LIN {X 0,Y 453.564,Z 567.99,A -85,B 0,C 180,E1 -8448.379,E2 -8448.379} C_VEL
LIN {X 0,Y 453.656,Z 567.978,A -85,B 0,C 180,E1 -8451.985,E2 -8451.985} C_VEL
LIN {X 0,Y 453.675,Z 567.975,A -85,B 0,C 180,E1 -8454.666,E2 -8454.666} C_VEL
LIN {X 0,Y 453.747,Z 567.964,A -85,B 0,C 180,E1 -8457.336,E2 -8457.336} C_VEL
LIN {X 0,Y 453.828,Z 567.956,A -85,B 0,C 180,E1 -8460,E2 -8460} C_VEL
LIN {X 0,Y 453.747,Z 567.966,A -85,B 0,C 180,E1 -8462.663,E2 -8462.663} C_VEL
LIN {X 0,Y 453.681,Z 567.975,A -85,B 0,C 180,E1 -8466.225,E2 -8466.225} C_VEL
LIN {X 0,Y 453.595,Z 567.985,A -85,B 0,C 180,E1 -8468.913,E2 -8468.913} C_VEL
LIN {X 0,Y 453.567,Z 567.989,A -85,B 0,C 180,E1 -8472.528,E2 -8472.528} C_VEL
LIN {X 0,Y 453.548,Z 567.991,A -85,B 0,C 180,E1 -8476.195,E2 -8476.195} C_VEL
LIN {X 0,Y 453.523,Z 567.992,A -85,B 0,C 180,E1 -8479.04,E2 -8479.04} C_VEL
LIN {X 0,Y 453.48,Z 567.998,A -85,B 0,C 180,E1 -8481.836,E2 -8481.836} C_VEL
LIN {X 0,Y 453.517,Z 567.995,A -85,B 0,C 180,E1 -8484.734,E2 -8484.734} C_VEL
LIN {X 0,Y 453.534,Z 567.991,A -85,B 0,C 180,E1 -8487.959,E2 -8487.959} C_VEL
LIN {X 0,Y 453.468,Z 567.999,A -85,B 0,C 180,E1 -8491.525,E2 -8491.525} C_VEL
LIN {X 0,Y 453.491,Z 567.999,A -85,B 0,C 180,E1 -8494.777,E2 -8494.777} C_VEL
LIN {X 0,Y 453.475,Z 568,A -85,B 0,C 180,E1 -8498.31,E2 -8498.31} C_VEL
LIN {X 0,Y 453.496,Z 567.998,A -85,B 0,C 180,E1 -8500.608,E2 -8500.608} C_VEL
LIN {X 0,Y 453.464,Z 568,A -85,B 0,C 180,E1 -8503.245,E2 -8503.245} C_VEL
LIN {X 0,Y 453.474,Z 567.999,A -85,B 0,C 180,E1 -8505.779,E2 -8505.779} C_VEL
LIN {X 0,Y 453.483,Z 568,A -85,B 0,C 180,E1 -8508.209,E2 -8508.209} C_VEL
LIN {X 0,Y 453.516,Z 567.995,A -85,B 0,C 180,E1 -8510.789,E2 -8510.789} C_VEL
LIN {X 0,Y 453.455,Z 568.002,A -85,B 0,C 180,E1 -8513.917,E2 -8513.917} C_VEL
LIN {X 0,Y 453.484,Z 567.998,A -85,B 0,C 180,E1 -8517.151,E2 -8517.151} C_VEL
LIN {X 0,Y 453.476,Z 568,A -85,B 0,C 180,E1 -8520.268,E2 -8520.268} C_VEL
LIN {X 0,Y 453.507,Z 567.994,A -85,B 0,C 180,E1 -8523.293,E2 -8523.293} C_VEL
LIN {X 0,Y 453.504,Z 567.996,A -85,B 0,C 180,E1 -8526.238,E2 -8526.238} C_VEL
LIN {X 0,Y 453.483,Z 567.997,A -85,B 0,C 180,E1 -8529.117,E2 -8529.117} C_VEL
LIN {X 0,Y 453.512,Z 567.994,A -85,B 0,C 180,E1 -8531.944,E2 -8531.944} C_VEL
LIN {X 0,Y 453.54,Z 567.993,A -85,B 0,C 180,E1 -8534.726,E2 -8534.726} C_VEL
LIN {X 0,Y 453.602,Z 567.981,A -85,B 0,C 180,E1 -8537.472,E2 -8537.472} C_VEL
LIN {X 0,Y 453.592,Z 567.984,A -85,B 0,C 180,E1 -8541.086,E2 -8541.086} C_VEL
LIN {X 0,Y 453.636,Z 567.979,A -85,B 0,C 180,E1 -8543.088,E2 -8543.088} C_VEL
LIN {X 0,Y 452.951,Z 568.063,A -85,B 0,C 180,E1 -8543.829,E2 -8543.829} C_VEL
LIN {X 0,Y 450.004,Z 568.433,A -85,B 0,C 180,E1 -8545.03,E2 -8545.03} C_VEL
LIN {X 0,Y 447.581,Z 568.733,A -85,B 0,C 180,E1 -8546,E2 -8546} C_VEL
LIN {X 0,Y 446.644,Z 568.851,A -85,B 0,C 180,E1 -8546.75,E2 -8546.75} C_VEL
LIN {X 0,Y 446.624,Z 568.852,A -85,B 0,C 180,E1 -8547.003,E2 -8547.003} C_VEL
LIN {X 0,Y 446.664,Z 568.85,A -85,B 0,C 180,E1 -8548.788,E2 -8548.788} C_VEL
LIN {X 0,Y 449.805,Z 580.017,A -85,B 0,C 180,E1 -8549.513,E2 -8549.513} C_VEL
LIN {X 0,Y 449.441,Z 591.841,A -85,B 0,C 180,E1 -8550.335,E2 -8550.335} C_VEL
LIN {X 0,Y 448.91,Z 603.225,A -85,B 0,C 180,E1 -8551.345,E2 -8551.345} C_VEL
LIN {X 0,Y 448.421,Z 613.322,A -85,B 0,C 180,E1 -8552.469,E2 -8552.469} C_VEL
LIN {X 0,Y 447.913,Z 621.552,A -85,B 0,C 180,E1 -8553.598,E2 -8553.598} C_VEL
LIN {X 0,Y 447.533,Z 629.569,A -85,B 0,C 180,E1 -8554.954,E2 -8554.954} C_VEL
LIN {X 0,Y 447.143,Z 636.058,A -85,B 0,C 180,E1 -8556.316,E2 -8556.316} C_VEL
LIN {X 0,Y 446.834,Z 641.437,A -85,B 0,C 180,E1 -8557.742,E2 -8557.742} C_VEL
LIN {X 0,Y 446.59,Z 645.265,A -85,B 0,C 180,E1 -8559.053,E2 -8559.053} C_VEL
LIN {X 0,Y 446.453,Z 647.36,A -85,B 0,C 180,E1 -8559.971,E2 -8559.971} C_VEL
LIN {X 0,Y 446.353,Z 649.018,A -85,B 0,C 180,E1 -8560.89,E2 -8560.89} C_VEL
LIN {X 0,Y 446.299,Z 650.921,A -85,B 0,C 180,E1 -8562.492,E2 -8562.492} C_VEL
LIN {X 0,Y 446.245,Z 651.532,A -85,B 0,C 180,E1 -8563.664,E2 -8563.664} C_VEL
LIN {X 0,Y 446.252,Z 651.557,A -85,B 0,C 180,E1 -8564.594,E2 -8564.594} C_VEL
LIN {X 0,Y 446.31,Z 650.697,A -85,B 0,C 180,E1 -8566.147,E2 -8566.147} C_VEL
LIN {X 0,Y 446.425,Z 649.136,A -85,B 0,C 180,E1 -8567.403,E2 -8567.403} C_VEL
LIN {X 0,Y 446.647,Z 646.444,A -85,B 0,C 180,E1 -8568.817,E2 -8568.817} C_VEL
LIN {X 0,Y 446.924,Z 642.659,A -85,B 0,C 180,E1 -8570.239,E2 -8570.239} C_VEL
LIN {X 0,Y 447.293,Z 637.798,A -85,B 0,C 180,E1 -8571.628,E2 -8571.628} C_VEL
LIN {X 0,Y 447.742,Z 631.225,A -85,B 0,C 180,E1 -8573.104,E2 -8573.104} C_VEL
LIN {X 0,Y 448.255,Z 623.531,A -85,B 0,C 180,E1 -8574.464,E2 -8574.464} C_VEL
LIN {X 0,Y 448.831,Z 614.481,A -85,B 0,C 180,E1 -8575.754,E2 -8575.754} C_VEL
LIN {X 0,Y 449.316,Z 605.52,A -85,B 0,C 180,E1 -8576.794,E2 -8576.794} C_VEL
LIN {X 0,Y 449.889,Z 594.487,A -85,B 0,C 180,E1 -8577.819,E2 -8577.819} C_VEL
LIN {X 0,Y 450.386,Z 583.545,A -85,B 0,C 180,E1 -8578.623,E2 -8578.623} C_VEL
LIN {X 0,Y 450.185,Z 580.766,A -85,B 0,C 180,E1 -8578.815,E2 -8578.815} C_VEL
LIN {X 0,Y 446.477,Z 568.873,A -85,B 0,C 180,E1 -8579.658,E2 -8579.658} C_VEL
LIN {X 0,Y 446.441,Z 568.875,A -85,B 0,C 180,E1 -8583.433,E2 -8583.433} C_VEL
LIN {X 0,Y 446.403,Z 568.88,A -85,B 0,C 180,E1 -8586.744,E2 -8586.744} C_VEL
LIN {X 0,Y 446.541,Z 568.984,A -85,B 0,C 180,E1 -8589.225,E2 -8589.225} C_VEL
LIN {X 0,Y 447.24,Z 574.12,A -85,B 0,C 180,E1 -8591.298,E2 -8591.298} C_VEL
LIN {X 0,Y 447.249,Z 580.496,A -85,B 0,C 180,E1 -8593.74,E2 -8593.74} C_VEL
LIN {X 0,Y 447.123,Z 588.594,A -85,B 0,C 180,E1 -8596.89,E2 -8596.89} C_VEL
LIN {X 0,Y 446.912,Z 596.265,A -85,B 0,C 180,E1 -8599.853,E2 -8599.853} C_VEL
LIN {X 0,Y 446.725,Z 605.271,A -85,B 0,C 180,E1 -8603.353,E2 -8603.353} C_VEL
LIN {X 0,Y 446.544,Z 613.573,A -85,B 0,C 180,E1 -8606.575,E2 -8606.575} C_VEL
LIN {X 0,Y 446.307,Z 622.453,A -85,B 0,C 180,E1 -8610.004,E2 -8610.004} C_VEL
LIN {X 0,Y 446.236,Z 624.977,A -85,B 0,C 180,E1 -8610.976,E2 -8610.976} C_VEL
LIN {X 0,Y 449.21,Z 639.613,A -85,B 0,C 180,E1 -8611.527,E2 -8611.527} C_VEL
LIN {X 0,Y 449.535,Z 644.304,A -85,B 0,C 180,E1 -8611.73,E2 -8611.73} C_VEL
LIN {X 0,Y 449.015,Z 657.282,A -85,B 0,C 180,E1 -8612.375,E2 -8612.375} C_VEL
LIN {X 0,Y 448.478,Z 669.514,A -85,B 0,C 180,E1 -8613.194,E2 -8613.194} C_VEL
LIN {X 0,Y 447.866,Z 681.12,A -85,B 0,C 180,E1 -8614.186,E2 -8614.186} C_VEL
LIN {X 0,Y 447.344,Z 691.417,A -85,B 0,C 180,E1 -8615.297,E2 -8615.297} C_VEL
LIN {X 0,Y 446.798,Z 701.201,A -85,B 0,C 180,E1 -8616.599,E2 -8616.599} C_VEL
LIN {X 0,Y 446.359,Z 708.49,A -85,B 0,C 180,E1 -8617.798,E2 -8617.798} C_VEL
LIN {X 0,Y 446.033,Z 715.547,A -85,B 0,C 180,E1 -8619.236,E2 -8619.236} C_VEL
LIN {X 0,Y 445.798,Z 721.109,A -85,B 0,C 180,E1 -8620.667,E2 -8620.667} C_VEL
LIN {X 0,Y 445.598,Z 725.362,A -85,B 0,C 180,E1 -8622.088,E2 -8622.088} C_VEL
LIN {X 0,Y 445.474,Z 728.448,A -85,B 0,C 180,E1 -8623.503,E2 -8623.503} C_VEL
LIN {X 0,Y 445.416,Z 729.89,A -85,B 0,C 180,E1 -8624.441,E2 -8624.441} C_VEL
LIN {X 0,Y 445.351,Z 730.909,A -85,B 0,C 180,E1 -8625.375,E2 -8625.375} C_VEL
LIN {X 0,Y 445.332,Z 731.517,A -85,B 0,C 180,E1 -8626.307,E2 -8626.307} C_VEL
LIN {X 0,Y 445.437,Z 731.452,A -85,B 0,C 180,E1 -8628.014,E2 -8628.014} C_VEL
LIN {X 0,Y 445.452,Z 730.713,A -85,B 0,C 180,E1 -8629.087,E2 -8629.087} C_VEL
LIN {X 0,Y 445.424,Z 729.609,A -85,B 0,C 180,E1 -8630.005,E2 -8630.005} C_VEL
LIN {X 0,Y 445.506,Z 728.063,A -85,B 0,C 180,E1 -8630.924,E2 -8630.924} C_VEL
LIN {X 0,Y 445.714,Z 724.923,A -85,B 0,C 180,E1 -8632.298,E2 -8632.298} C_VEL
LIN {X 0,Y 445.881,Z 720.726,A -85,B 0,C 180,E1 -8633.666,E2 -8633.666} C_VEL
LIN {X 0,Y 446.089,Z 715.369,A -85,B 0,C 180,E1 -8635.029,E2 -8635.029} C_VEL
LIN {X 0,Y 446.421,Z 708.676,A -85,B 0,C 180,E1 -8636.39,E2 -8636.39} C_VEL
LIN {X 0,Y 446.93,Z 700.288,A -85,B 0,C 180,E1 -8637.747,E2 -8637.747} C_VEL
LIN {X 0,Y 447.442,Z 691.738,A -85,B 0,C 180,E1 -8638.875,E2 -8638.875} C_VEL
LIN {X 0,Y 448.043,Z 681.265,A -85,B 0,C 180,E1 -8640,E2 -8640} C_VEL
LIN {X 0,Y 448.704,Z 669.341,A -85,B 0,C 180,E1 -8641.01,E2 -8641.01} C_VEL
LIN {X 0,Y 449.223,Z 657.538,A -85,B 0,C 180,E1 -8641.793,E2 -8641.793} C_VEL
LIN {X 0,Y 449.771,Z 643.87,A -85,B 0,C 180,E1 -8642.463,E2 -8642.463} C_VEL
LIN {X 0,Y 449.345,Z 639.264,A -85,B 0,C 180,E1 -8642.662,E2 -8642.662} C_VEL
LIN {X 0,Y 446.397,Z 626.394,A -85,B 0,C 180,E1 -8643.187,E2 -8643.187} C_VEL
LIN {X 0,Y 446.599,Z 619.374,A -85,B 0,C 180,E1 -8645.871,E2 -8645.871} C_VEL
LIN {X 0,Y 446.8,Z 611.001,A -85,B 0,C 180,E1 -8649.05,E2 -8649.05} C_VEL
LIN {X 0,Y 446.991,Z 602.445,A -85,B 0,C 180,E1 -8652.255,E2 -8652.255} C_VEL
LIN {X 0,Y 447.091,Z 594.826,A -85,B 0,C 180,E1 -8655.033,E2 -8655.033} C_VEL
LIN {X 0,Y 447.176,Z 586.88,A -85,B 0,C 180,E1 -8657.847,E2 -8657.847} C_VEL
LIN {X 0,Y 447.237,Z 578.64,A -85,B 0,C 180,E1 -8660.706,E2 -8660.706} C_VEL
LIN {X 0,Y 447.122,Z 572.869,A -85,B 0,C 180,E1 -8662.65,E2 -8662.65} C_VEL
LIN {X 0,Y 446.461,Z 568.878,A -85,B 0,C 180,E1 -8664.078,E2 -8664.078} C_VEL
LIN {X 0,Y 446.475,Z 568.874,A -85,B 0,C 180,E1 -8667.161,E2 -8667.161} C_VEL
LIN {X 0,Y 446.43,Z 568.878,A -85,B 0,C 180,E1 -8670.25,E2 -8670.25} C_VEL
LIN {X 0,Y 446.439,Z 568.878,A -85,B 0,C 180,E1 -8673.455,E2 -8673.455} C_VEL
LIN {X 0,Y 446.405,Z 568.88,A -85,B 0,C 180,E1 -8676.745,E2 -8676.745} C_VEL
LIN {X 0,Y 446.486,Z 568.871,A -85,B 0,C 180,E1 -8679.532,E2 -8679.532} C_VEL
LIN {X 0,Y 446.446,Z 568.872,A -85,B 0,C 180,E1 -8682.603,E2 -8682.603} C_VEL
LIN {X 0,Y 446.454,Z 568.873,A -85,B 0,C 180,E1 -8685.104,E2 -8685.104} C_VEL
LIN {X 0,Y 446.473,Z 568.88,A -85,B 0,C 180,E1 -8688.082,E2 -8688.082} C_VEL
LIN {X 0,Y 448.181,Z 577.008,A -85,B 0,C 180,E1 -8690.723,E2 -8690.723} C_VEL
LIN {X 0,Y 449.575,Z 585.238,A -85,B 0,C 180,E1 -8693.23,E2 -8693.23} C_VEL
LIN {X 0,Y 449.259,Z 592.261,A -85,B 0,C 180,E1 -8695.182,E2 -8695.182} C_VEL
LIN {X 0,Y 448.477,Z 604.164,A -85,B 0,C 180,E1 -8698.335,E2 -8698.335} C_VEL
LIN {X 0,Y 447.866,Z 616.519,A -85,B 0,C 180,E1 -8701.494,E2 -8701.494} C_VEL
LIN {X 0,Y 447.316,Z 629.239,A -85,B 0,C 180,E1 -8704.652,E2 -8704.652} C_VEL
LIN {X 0,Y 446.848,Z 642.343,A -85,B 0,C 180,E1 -8707.824,E2 -8707.824} C_VEL
LIN {X 0,Y 446.454,Z 656.717,A -85,B 0,C 180,E1 -8711.236,E2 -8711.236} C_VEL
LIN {X 0,Y 446.199,Z 667.476,A -85,B 0,C 180,E1 -8713.76,E2 -8713.76} C_VEL
LIN {X 0,Y 447.644,Z 682.292,A -85,B 0,C 180,E1 -8714.193,E2 -8714.193} C_VEL
LIN {X 0,Y 448.622,Z 693.605,A -85,B 0,C 180,E1 -8714.672,E2 -8714.672} C_VEL
LIN {X 0,Y 448.942,Z 698.381,A -85,B 0,C 180,E1 -8714.916,E2 -8714.916} C_VEL
LIN {X 0,Y 448.329,Z 710.074,A -85,B 0,C 180,E1 -8715.591,E2 -8715.591} C_VEL
LIN {X 0,Y 447.513,Z 725.482,A -85,B 0,C 180,E1 -8716.737,E2 -8716.737} C_VEL
LIN {X 0,Y 447.06,Z 736.228,A -85,B 0,C 180,E1 -8717.748,E2 -8717.748} C_VEL
LIN {X 0,Y 446.662,Z 744.258,A -85,B 0,C 180,E1 -8718.658,E2 -8718.658} C_VEL
LIN {X 0,Y 446.157,Z 754.155,A -85,B 0,C 180,E1 -8720.023,E2 -8720.023} C_VEL
LIN {X 0,Y 445.918,Z 762.062,A -85,B 0,C 180,E1 -8721.39,E2 -8721.39} C_VEL
LIN {X 0,Y 445.702,Z 768.393,A -85,B 0,C 180,E1 -8722.754,E2 -8722.754} C_VEL
LIN {X 0,Y 445.61,Z 773.404,A -85,B 0,C 180,E1 -8724.117,E2 -8724.117} C_VEL
LIN {X 0,Y 445.549,Z 777.237,A -85,B 0,C 180,E1 -8725.477,E2 -8725.477} C_VEL
LIN {X 0,Y 445.576,Z 779.215,A -85,B 0,C 180,E1 -8726.384,E2 -8726.384} C_VEL
LIN {X 0,Y 445.559,Z 780.717,A -85,B 0,C 180,E1 -8727.289,E2 -8727.289} C_VEL
LIN {X 0,Y 445.587,Z 781.784,A -85,B 0,C 180,E1 -8728.193,E2 -8728.193} C_VEL
LIN {X 0,Y 445.533,Z 782.44,A -85,B 0,C 180,E1 -8729.097,E2 -8729.097} C_VEL
LIN {X 0,Y 445.518,Z 782.686,A -85,B 0,C 180,E1 -8730.001,E2 -8730.001} C_VEL
LIN {X 0,Y 445.532,Z 782.478,A -85,B 0,C 180,E1 -8730.905,E2 -8730.905} C_VEL
LIN {X 0,Y 445.589,Z 781.868,A -85,B 0,C 180,E1 -8731.808,E2 -8731.808} C_VEL
LIN {X 0,Y 445.559,Z 780.849,A -85,B 0,C 180,E1 -8732.713,E2 -8732.713} C_VEL
LIN {X 0,Y 445.557,Z 779.38,A -85,B 0,C 180,E1 -8733.618,E2 -8733.618} C_VEL
LIN {X 0,Y 445.587,Z 776.336,A -85,B 0,C 180,E1 -8734.977,E2 -8734.977} C_VEL
LIN {X 0,Y 445.606,Z 771.713,A -85,B 0,C 180,E1 -8736.472,E2 -8736.472} C_VEL
LIN {X 0,Y 445.775,Z 765.814,A -85,B 0,C 180,E1 -8737.93,E2 -8737.93} C_VEL
LIN {X 0,Y 446.057,Z 758.843,A -85,B 0,C 180,E1 -8739.295,E2 -8739.295} C_VEL
LIN {X 0,Y 446.369,Z 750.055,A -85,B 0,C 180,E1 -8740.662,E2 -8740.662} C_VEL
LIN {X 0,Y 446.882,Z 740.065,A -85,B 0,C 180,E1 -8741.913,E2 -8741.913} C_VEL
LIN {X 0,Y 447.402,Z 729.917,A -85,B 0,C 180,E1 -8742.931,E2 -8742.931} C_VEL
LIN {X 0,Y 447.941,Z 718.601,A -85,B 0,C 180,E1 -8743.844,E2 -8743.844} C_VEL
LIN {X 0,Y 448.662,Z 703.299,A -85,B 0,C 180,E1 -8744.805,E2 -8744.805} C_VEL
LIN {X 0,Y 448.802,Z 695.545,A -85,B 0,C 180,E1 -8745.207,E2 -8745.207} C_VEL
LIN {X 0,Y 447.666,Z 683.767,A -85,B 0,C 180,E1 -8745.715,E2 -8745.715} C_VEL
LIN {X 0,Y 446.358,Z 670.167,A -85,B 0,C 180,E1 -8746.115,E2 -8746.115} C_VEL
LIN {X 0,Y 446.199,Z 668.118,A -85,B 0,C 180,E1 -8746.167,E2 -8746.167} C_VEL
LIN {X 0,Y 446.509,Z 654.736,A -85,B 0,C 180,E1 -8749.302,E2 -8749.302} C_VEL
LIN {X 0,Y 446.896,Z 640.552,A -85,B 0,C 180,E1 -8752.663,E2 -8752.663} C_VEL
LIN {X 0,Y 447.412,Z 626.287,A -85,B 0,C 180,E1 -8756.094,E2 -8756.094} C_VEL
LIN {X 0,Y 447.957,Z 612.97,A -85,B 0,C 180,E1 -8759.36,E2 -8759.36} C_VEL
LIN {X 0,Y 448.613,Z 599.587,A -85,B 0,C 180,E1 -8762.716,E2 -8762.716} C_VEL
LIN {X 0,Y 449.258,Z 587.106,A -85,B 0,C 180,E1 -8765.954,E2 -8765.954} C_VEL
LIN {X 0,Y 449.03,Z 582.145,A -85,B 0,C 180,E1 -8767.295,E2 -8767.295} C_VEL
LIN {X 0,Y 446.799,Z 570.625,A -85,B 0,C 180,E1 -8770.649,E2 -8770.649} C_VEL
LIN {X 0,Y 446.461,Z 568.874,A -85,B 0,C 180,E1 -8771.187,E2 -8771.187} C_VEL
LIN {X 0,Y 446.458,Z 568.874,A -85,B 0,C 180,E1 -8774.897,E2 -8774.897} C_VEL
LIN {X 0,Y 446.433,Z 568.877,A -85,B 0,C 180,E1 -8778.609,E2 -8778.609} C_VEL
LIN {X 0,Y 446.465,Z 568.872,A -85,B 0,C 180,E1 -8780.975,E2 -8780.975} C_VEL
LIN {X 0,Y 446.426,Z 568.878,A -85,B 0,C 180,E1 -8784.374,E2 -8784.374} C_VEL
LIN {X 0,Y 446.427,Z 568.877,A -85,B 0,C 180,E1 -8787.638,E2 -8787.638} C_VEL
LIN {X 0,Y 446.453,Z 568.874,A -85,B 0,C 180,E1 -8790.791,E2 -8790.791} C_VEL
LIN {X 0,Y 446.483,Z 568.87,A -85,B 0,C 180,E1 -8793.848,E2 -8793.848} C_VEL
LIN {X 0,Y 446.433,Z 568.876,A -85,B 0,C 180,E1 -8796.823,E2 -8796.823} C_VEL
LIN {X 0,Y 446.449,Z 568.873,A -85,B 0,C 180,E1 -8799.737,E2 -8799.737} C_VEL
LIN {X 0,Y 446.468,Z 568.873,A -85,B 0,C 180,E1 -8802.597,E2 -8802.597} C_VEL
LIN {X 0,Y 446.474,Z 568.869,A -85,B 0,C 180,E1 -8805.412,E2 -8805.412} C_VEL
LIN {X 0,Y 446.522,Z 568.867,A -85,B 0,C 180,E1 -8808.193,E2 -8808.193} C_VEL
LIN {X 0,Y 446.605,Z 568.855,A -85,B 0,C 180,E1 -8811.858,E2 -8811.858} C_VEL
LIN {X 0,Y 446.649,Z 568.85,A -85,B 0,C 180,E1 -8814.582,E2 -8814.582} C_VEL
LIN {X 0,Y 446.667,Z 568.848,A -85,B 0,C 180,E1 -8818.196,E2 -8818.196} C_VEL
LIN {X 0,Y 446.798,Z 568.831,A -85,B 0,C 180,E1 -8820,E2 -8820} C_VEL
LIN {X 0,Y 446.694,Z 568.844,A -85,B 0,C 180,E1 -8822.705,E2 -8822.705} C_VEL
LIN {X 0,Y 446.65,Z 568.851,A -85,B 0,C 180,E1 -8826.323,E2 -8826.323} C_VEL
LIN {X 0,Y 446.541,Z 568.863,A -85,B 0,C 180,E1 -8829.055,E2 -8829.055} C_VEL
LIN {X 0,Y 446.525,Z 568.866,A -85,B 0,C 180,E1 -8832.729,E2 -8832.729} C_VEL
LIN {X 0,Y 446.499,Z 568.869,A -85,B 0,C 180,E1 -8836.227,E2 -8836.227} C_VEL
LIN {X 0,Y 446.472,Z 568.87,A -85,B 0,C 180,E1 -8839.303,E2 -8839.303} C_VEL
LIN {X 0,Y 446.422,Z 568.879,A -85,B 0,C 180,E1 -8842.199,E2 -8842.199} C_VEL
LIN {X 0,Y 446.46,Z 568.872,A -85,B 0,C 180,E1 -8845.152,E2 -8845.152} C_VEL
LIN {X 0,Y 446.487,Z 568.871,A -85,B 0,C 180,E1 -8848.178,E2 -8848.178} C_VEL
LIN {X 0,Y 446.421,Z 568.877,A -85,B 0,C 180,E1 -8851.774,E2 -8851.774} C_VEL
LIN {X 0,Y 446.432,Z 568.878,A -85,B 0,C 180,E1 -8854.522,E2 -8854.522} C_VEL
LIN {X 0,Y 446.432,Z 568.877,A -85,B 0,C 180,E1 -8858.081,E2 -8858.081} C_VEL
LIN {X 0,Y 446.429,Z 568.877,A -85,B 0,C 180,E1 -8860.917,E2 -8860.917} C_VEL
LIN {X 0,Y 446.424,Z 568.877,A -85,B 0,C 180,E1 -8863.843,E2 -8863.843} C_VEL
LIN {X 0,Y 446.422,Z 568.879,A -85,B 0,C 180,E1 -8866.4,E2 -8866.4} C_VEL
LIN {X 0,Y 446.452,Z 568.872,A -85,B 0,C 180,E1 -8869.802,E2 -8869.802} C_VEL
LIN {X 0,Y 446.41,Z 568.879,A -85,B 0,C 180,E1 -8872.121,E2 -8872.121} C_VEL
LIN {X 0,Y 446.429,Z 568.874,A -85,B 0,C 180,E1 -8875.476,E2 -8875.476} C_VEL
LIN {X 0,Y 446.417,Z 568.879,A -85,B 0,C 180,E1 -8878.699,E2 -8878.699} C_VEL
LIN {X 0,Y 446.485,Z 568.869,A -85,B 0,C 180,E1 -8881.821,E2 -8881.821} C_VEL
LIN {X 0,Y 446.458,Z 568.874,A -85,B 0,C 180,E1 -8884.847,E2 -8884.847} C_VEL
LIN {X 0,Y 446.448,Z 568.875,A -85,B 0,C 180,E1 -8888.244,E2 -8888.244} C_VEL
LIN {X 0,Y 446.457,Z 568.872,A -85,B 0,C 180,E1 -8891.648,E2 -8891.648} C_VEL
LIN {X 0,Y 446.507,Z 568.868,A -85,B 0,C 180,E1 -8894.479,E2 -8894.479} C_VEL
LIN {X 0,Y 446.539,Z 568.863,A -85,B 0,C 180,E1 -8898.193,E2 -8898.193} C_VEL
LIN {X 0,Y 446.599,Z 568.855,A -85,B 0,C 180,E1 -8901.857,E2 -8901.857} C_VEL
LIN {X 0,Y 446.646,Z 568.851,A -85,B 0,C 180,E1 -8904.582,E2 -8904.582} C_VEL
LIN {X 0,Y 446.624,Z 568.852,A -85,B 0,C 180,E1 -8907.003,E2 -8907.003} C_VEL
LIN {X 0,Y 446.545,Z 569.451,A -85,B 0,C 180,E1 -8907.484,E2 -8907.484} C_VEL
LIN {X 0,Y 446.018,Z 571.501,A -85,B 0,C 180,E1 -8908.037,E2 -8908.037} C_VEL
LIN {X 0,Y 445.228,Z 574.508,A -85,B 0,C 180,E1 -8908.524,E2 -8908.524} C_VEL
LIN {X 0,Y 444.132,Z 579.092,A -85,B 0,C 180,E1 -8909.036,E2 -8909.036} C_VEL
LIN {X 0,Y 442.942,Z 586.043,A -85,B 0,C 180,E1 -8909.63,E2 -8909.63} C_VEL
LIN {X 0,Y 442.691,Z 589.675,A -85,B 0,C 180,E1 -8909.904,E2 -8909.904} C_VEL
LIN {X 0,Y 442.248,Z 600.357,A -85,B 0,C 180,E1 -8910.796,E2 -8910.796} C_VEL
LIN {X 0,Y 441.688,Z 610.257,A -85,B 0,C 180,E1 -8911.823,E2 -8911.823} C_VEL
LIN {X 0,Y 441.241,Z 619.171,A -85,B 0,C 180,E1 -8912.966,E2 -8912.966} C_VEL
LIN {X 0,Y 440.688,Z 627.905,A -85,B 0,C 180,E1 -8914.344,E2 -8914.344} C_VEL
LIN {X 0,Y 440.327,Z 634.909,A -85,B 0,C 180,E1 -8915.724,E2 -8915.724} C_VEL
LIN {X 0,Y 439.934,Z 641.307,A -85,B 0,C 180,E1 -8917.342,E2 -8917.342} C_VEL
LIN {X 0,Y 439.637,Z 645.554,A -85,B 0,C 180,E1 -8918.734,E2 -8918.734} C_VEL
LIN {X 0,Y 439.41,Z 648.748,A -85,B 0,C 180,E1 -8920.132,E2 -8920.132} C_VEL
LIN {X 0,Y 439.319,Z 650.338,A -85,B 0,C 180,E1 -8921.067,E2 -8921.067} C_VEL
LIN {X 0,Y 439.263,Z 652.015,A -85,B 0,C 180,E1 -8922.587,E2 -8922.587} C_VEL
LIN {X 0,Y 439.23,Z 652.584,A -85,B 0,C 180,E1 -8923.886,E2 -8923.886} C_VEL
LIN {X 0,Y 439.244,Z 652.544,A -85,B 0,C 180,E1 -8924.832,E2 -8924.832} C_VEL
LIN {X 0,Y 439.32,Z 651.643,A -85,B 0,C 180,E1 -8926.293,E2 -8926.293} C_VEL
LIN {X 0,Y 439.475,Z 649.847,A -85,B 0,C 180,E1 -8927.688,E2 -8927.688} C_VEL
LIN {X 0,Y 439.605,Z 648.077,A -85,B 0,C 180,E1 -8928.646,E2 -8928.646} C_VEL
LIN {X 0,Y 439.924,Z 644.505,A -85,B 0,C 180,E1 -8930.088,E2 -8930.088} C_VEL
LIN {X 0,Y 440.279,Z 639.729,A -85,B 0,C 180,E1 -8931.538,E2 -8931.538} C_VEL
LIN {X 0,Y 440.736,Z 633.578,A -85,B 0,C 180,E1 -8932.996,E2 -8932.996} C_VEL
LIN {X 0,Y 441.311,Z 625.787,A -85,B 0,C 180,E1 -8934.459,E2 -8934.459} C_VEL
LIN {X 0,Y 441.85,Z 617.635,A -85,B 0,C 180,E1 -8935.685,E2 -8935.685} C_VEL
LIN {X 0,Y 442.496,Z 607.184,A -85,B 0,C 180,E1 -8936.952,E2 -8936.952} C_VEL
LIN {X 0,Y 443.025,Z 597.455,A -85,B 0,C 180,E1 -8937.902,E2 -8937.902} C_VEL
LIN {X 0,Y 443.568,Z 586.75,A -85,B 0,C 180,E1 -8938.737,E2 -8938.737} C_VEL
LIN {X 0,Y 443.546,Z 582.847,A -85,B 0,C 180,E1 -8939.006,E2 -8939.006} C_VEL
LIN {X 0,Y 440.116,Z 572.057,A -85,B 0,C 180,E1 -8939.796,E2 -8939.796} C_VEL
LIN {X 0,Y 439.406,Z 569.754,A -85,B 0,C 180,E1 -8939.964,E2 -8939.964} C_VEL
LIN {X 0,Y 439.367,Z 569.758,A -85,B 0,C 180,E1 -8942.945,E2 -8942.945} C_VEL
LIN {X 0,Y 439.37,Z 569.758,A -85,B 0,C 180,E1 -8946.286,E2 -8946.286} C_VEL
LIN {X 0,Y 439.449,Z 569.817,A -85,B 0,C 180,E1 -8949.028,E2 -8949.028} C_VEL
LIN {X 0,Y 440.298,Z 575.715,A -85,B 0,C 180,E1 -8951.392,E2 -8951.392} C_VEL
LIN {X 0,Y 440.23,Z 582.535,A -85,B 0,C 180,E1 -8954.078,E2 -8954.078} C_VEL
LIN {X 0,Y 440.107,Z 590.752,A -85,B 0,C 180,E1 -8957.269,E2 -8957.269} C_VEL
LIN {X 0,Y 439.843,Z 598.463,A -85,B 0,C 180,E1 -8960.273,E2 -8960.273} C_VEL
LIN {X 0,Y 439.732,Z 605.556,A -85,B 0,C 180,E1 -8963.044,E2 -8963.044} C_VEL
LIN {X 0,Y 439.507,Z 614.788,A -85,B 0,C 180,E1 -8966.653,E2 -8966.653} C_VEL
LIN {X 0,Y 439.291,Z 622.768,A -85,B 0,C 180,E1 -8969.757,E2 -8969.757} C_VEL
LIN {X 0,Y 439.233,Z 625.394,A -85,B 0,C 180,E1 -8970.743,E2 -8970.743} C_VEL
LIN {X 0,Y 442.097,Z 639.128,A -85,B 0,C 180,E1 -8971.258,E2 -8971.258} C_VEL
LIN {X 0,Y 442.687,Z 644.43,A -85,B 0,C 180,E1 -8971.494,E2 -8971.494} C_VEL
LIN {X 0,Y 442.151,Z 656.661,A -85,B 0,C 180,E1 -8972.102,E2 -8972.102} C_VEL
LIN {X 0,Y 441.631,Z 669.237,A -85,B 0,C 180,E1 -8972.945,E2 -8972.945} C_VEL
LIN {X 0,Y 441.008,Z 680.247,A -85,B 0,C 180,E1 -8973.881,E2 -8973.881} C_VEL
LIN {X 0,Y 440.435,Z 690.622,A -85,B 0,C 180,E1 -8974.985,E2 -8974.985} C_VEL
LIN {X 0,Y 439.899,Z 699.935,A -85,B 0,C 180,E1 -8976.209,E2 -8976.209} C_VEL
LIN {X 0,Y 439.403,Z 707.542,A -85,B 0,C 180,E1 -8977.427,E2 -8977.427} C_VEL
LIN {X 0,Y 439.079,Z 714.913,A -85,B 0,C 180,E1 -8978.892,E2 -8978.892} C_VEL
LIN {X 0,Y 438.767,Z 720.683,A -85,B 0,C 180,E1 -8980.345,E2 -8980.345} C_VEL
LIN {X 0,Y 438.537,Z 725.133,A -85,B 0,C 180,E1 -8981.79,E2 -8981.79} C_VEL
LIN {X 0,Y 438.41,Z 728.405,A -85,B 0,C 180,E1 -8983.229,E2 -8983.229} C_VEL
LIN {X 0,Y 438.354,Z 730.007,A -85,B 0,C 180,E1 -8984.184,E2 -8984.184} C_VEL
LIN {X 0,Y 438.289,Z 731.112,A -85,B 0,C 180,E1 -8985.134,E2 -8985.134} C_VEL
LIN {X 0,Y 438.26,Z 731.802,A -85,B 0,C 180,E1 -8986.082,E2 -8986.082} C_VEL
LIN {X 0,Y 438.254,Z 732.085,A -85,B 0,C 180,E1 -8987.026,E2 -8987.026} C_VEL
LIN {X 0,Y 438.364,Z 731.896,A -85,B 0,C 180,E1 -8987.971,E2 -8987.971} C_VEL
LIN {X 0,Y 438.359,Z 731.309,A -85,B 0,C 180,E1 -8988.908,E2 -8988.908} C_VEL
LIN {X 0,Y 438.344,Z 730.33,A -85,B 0,C 180,E1 -8989.842,E2 -8989.842} C_VEL
LIN {X 0,Y 438.418,Z 728.894,A -85,B 0,C 180,E1 -8990.776,E2 -8990.776} C_VEL
LIN {X 0,Y 438.634,Z 725.92,A -85,B 0,C 180,E1 -8992.173,E2 -8992.173} C_VEL
LIN {X 0,Y 438.814,Z 721.901,A -85,B 0,C 180,E1 -8993.563,E2 -8993.563} C_VEL
LIN {X 0,Y 439.019,Z 716.728,A -85,B 0,C 180,E1 -8994.949,E2 -8994.949} C_VEL
LIN {X 0,Y 439.362,Z 710.236,A -85,B 0,C 180,E1 -8996.332,E2 -8996.332} C_VEL
LIN {X 0,Y 439.896,Z 702.178,A -85,B 0,C 180,E1 -8997.711,E2 -8997.711} C_VEL
LIN {X 0,Y 440.415,Z 693.91,A -85,B 0,C 180,E1 -8998.857,E2 -8998.857} C_VEL
LIN {X 0,Y 441.052,Z 683.803,A -85,B 0,C 180,E1 -9000,E2 -9000} C_VEL
LIN {X 0,Y 441.625,Z 673.903,A -85,B 0,C 180,E1 -9000.912,E2 -9000.912} C_VEL
LIN {X 0,Y 442.17,Z 663.25,A -85,B 0,C 180,E1 -9001.708,E2 -9001.708} C_VEL
LIN {X 0,Y 442.782,Z 650.36,A -85,B 0,C 180,E1 -9002.445,E2 -9002.445} C_VEL
LIN {X 0,Y 442.81,Z 641.967,A -85,B 0,C 180,E1 -9002.829,E2 -9002.829} C_VEL
LIN {X 0,Y 440.489,Z 631.681,A -85,B 0,C 180,E1 -9003.287,E2 -9003.287} C_VEL
LIN {X 0,Y 439.341,Z 626.805,A -85,B 0,C 180,E1 -9003.497,E2 -9003.497} C_VEL
LIN {X 0,Y 439.601,Z 620.38,A -85,B 0,C 180,E1 -9005.965,E2 -9005.965} C_VEL
LIN {X 0,Y 439.833,Z 611.923,A -85,B 0,C 180,E1 -9009.195,E2 -9009.195} C_VEL
LIN {X 0,Y 440.051,Z 603.416,A -85,B 0,C 180,E1 -9012.451,E2 -9012.451} C_VEL
LIN {X 0,Y 440.174,Z 595.735,A -85,B 0,C 180,E1 -9015.275,E2 -9015.275} C_VEL
LIN {X 0,Y 440.235,Z 587.654,A -85,B 0,C 180,E1 -9018.138,E2 -9018.138} C_VEL
LIN {X 0,Y 440.317,Z 579.349,A -85,B 0,C 180,E1 -9021.047,E2 -9021.047} C_VEL
LIN {X 0,Y 440.122,Z 573.583,A -85,B 0,C 180,E1 -9023.031,E2 -9023.031} C_VEL
LIN {X 0,Y 439.416,Z 569.756,A -85,B 0,C 180,E1 -9024.371,E2 -9024.371} C_VEL
LIN {X 0,Y 439.438,Z 569.75,A -85,B 0,C 180,E1 -9027.633,E2 -9027.633} C_VEL
LIN {X 0,Y 439.361,Z 569.76,A -85,B 0,C 180,E1 -9030.789,E2 -9030.789} C_VEL
LIN {X 0,Y 439.382,Z 569.755,A -85,B 0,C 180,E1 -9034.045,E2 -9034.045} C_VEL
LIN {X 0,Y 439.359,Z 569.759,A -85,B 0,C 180,E1 -9037.435,E2 -9037.435} C_VEL
LIN {X 0,Y 439.423,Z 569.749,A -85,B 0,C 180,E1 -9039.854,E2 -9039.854} C_VEL
LIN {X 0,Y 439.399,Z 569.749,A -85,B 0,C 180,E1 -9042.631,E2 -9042.631} C_VEL
LIN {X 0,Y 439.4,Z 569.753,A -85,B 0,C 180,E1 -9046.035,E2 -9046.035} C_VEL
LIN {X 0,Y 439.449,Z 569.918,A -85,B 0,C 180,E1 -9047.75,E2 -9047.75} C_VEL
LIN {X 0,Y 441.439,Z 579.437,A -85,B 0,C 180,E1 -9050.898,E2 -9050.898} C_VEL
LIN {X 0,Y 442.582,Z 585.827,A -85,B 0,C 180,E1 -9052.886,E2 -9052.886} C_VEL
LIN {X 0,Y 442.56,Z 589.998,A -85,B 0,C 180,E1 -9054.086,E2 -9054.086} C_VEL
LIN {X 0,Y 441.754,Z 601.523,A -85,B 0,C 180,E1 -9057.255,E2 -9057.255} C_VEL
LIN {X 0,Y 441.067,Z 613.437,A -85,B 0,C 180,E1 -9060.4,E2 -9060.4} C_VEL
LIN {X 0,Y 440.435,Z 626.445,A -85,B 0,C 180,E1 -9063.718,E2 -9063.718} C_VEL
LIN {X 0,Y 439.871,Z 639.478,A -85,B 0,C 180,E1 -9066.957,E2 -9066.957} C_VEL
LIN {X 0,Y 439.42,Z 653.521,A -85,B 0,C 180,E1 -9070.376,E2 -9070.376} C_VEL
LIN {X 0,Y 439.162,Z 666.411,A -85,B 0,C 180,E1 -9073.469,E2 -9073.469} C_VEL
LIN {X 0,Y 440.643,Z 681.459,A -85,B 0,C 180,E1 -9073.923,E2 -9073.923} C_VEL
LIN {X 0,Y 441.661,Z 694.175,A -85,B 0,C 180,E1 -9074.484,E2 -9074.484} C_VEL
LIN {X 0,Y 441.998,Z 698.759,A -85,B 0,C 180,E1 -9074.732,E2 -9074.732} C_VEL
LIN {X 0,Y 441.32,Z 710.904,A -85,B 0,C 180,E1 -9075.475,E2 -9075.475} C_VEL
LIN {X 0,Y 440.681,Z 723.175,A -85,B 0,C 180,E1 -9076.366,E2 -9076.366} C_VEL
LIN {X 0,Y 440.212,Z 733.636,A -85,B 0,C 180,E1 -9077.32,E2 -9077.32} C_VEL
LIN {X 0,Y 439.671,Z 741.989,A -85,B 0,C 180,E1 -9078.241,E2 -9078.241} C_VEL
LIN {X 0,Y 439.28,Z 750.707,A -85,B 0,C 180,E1 -9079.399,E2 -9079.399} C_VEL
LIN {X 0,Y 438.945,Z 759.172,A -85,B 0,C 180,E1 -9080.788,E2 -9080.788} C_VEL
LIN {X 0,Y 438.711,Z 766.003,A -85,B 0,C 180,E1 -9082.175,E2 -9082.175} C_VEL
LIN {X 0,Y 438.517,Z 772.312,A -85,B 0,C 180,E1 -9083.817,E2 -9083.817} C_VEL
LIN {X 0,Y 438.471,Z 776.812,A -85,B 0,C 180,E1 -9085.404,E2 -9085.404} C_VEL
LIN {X 0,Y 438.476,Z 778.797,A -85,B 0,C 180,E1 -9086.325,E2 -9086.325} C_VEL
LIN {X 0,Y 438.482,Z 780.304,A -85,B 0,C 180,E1 -9087.245,E2 -9087.245} C_VEL
LIN {X 0,Y 438.494,Z 781.374,A -85,B 0,C 180,E1 -9088.164,E2 -9088.164} C_VEL
LIN {X 0,Y 438.466,Z 782.035,A -85,B 0,C 180,E1 -9089.082,E2 -9089.082} C_VEL
LIN {X 0,Y 438.449,Z 782.28,A -85,B 0,C 180,E1 -9090.001,E2 -9090.001} C_VEL
LIN {X 0,Y 438.466,Z 782.071,A -85,B 0,C 180,E1 -9090.919,E2 -9090.919} C_VEL
LIN {X 0,Y 438.496,Z 781.459,A -85,B 0,C 180,E1 -9091.838,E2 -9091.838} C_VEL
LIN {X 0,Y 438.481,Z 780.439,A -85,B 0,C 180,E1 -9092.757,E2 -9092.757} C_VEL
LIN {X 0,Y 438.458,Z 778.961,A -85,B 0,C 180,E1 -9093.677,E2 -9093.677} C_VEL
LIN {X 0,Y 438.516,Z 775.91,A -85,B 0,C 180,E1 -9095.058,E2 -9095.058} C_VEL
LIN {X 0,Y 438.525,Z 771.679,A -85,B 0,C 180,E1 -9096.463,E2 -9096.463} C_VEL
LIN {X 0,Y 438.715,Z 765.364,A -85,B 0,C 180,E1 -9098.059,E2 -9098.059} C_VEL
LIN {X 0,Y 438.991,Z 758.372,A -85,B 0,C 180,E1 -9099.446,E2 -9099.446} C_VEL
LIN {X 0,Y 439.354,Z 749.565,A -85,B 0,C 180,E1 -9100.834,E2 -9100.834} C_VEL
LIN {X 0,Y 439.845,Z 739.55,A -85,B 0,C 180,E1 -9102.106,E2 -9102.106} C_VEL
LIN {X 0,Y 440.381,Z 729.402,A -85,B 0,C 180,E1 -9103.139,E2 -9103.139} C_VEL
LIN {X 0,Y 441.017,Z 718.027,A -85,B 0,C 180,E1 -9104.066,E2 -9104.066} C_VEL
LIN {X 0,Y 441.562,Z 706.33,A -85,B 0,C 180,E1 -9104.813,E2 -9104.813} C_VEL
LIN {X 0,Y 441.859,Z 696.538,A -85,B 0,C 180,E1 -9105.334,E2 -9105.334} C_VEL
LIN {X 0,Y 440.792,Z 685.195,A -85,B 0,C 180,E1 -9105.861,E2 -9105.861} C_VEL
LIN {X 0,Y 439.613,Z 672.389,A -85,B 0,C 180,E1 -9106.287,E2 -9106.287} C_VEL
LIN {X 0,Y 439.152,Z 667.125,A -85,B 0,C 180,E1 -9106.414,E2 -9106.414} C_VEL
LIN {X 0,Y 439.459,Z 652.675,A -85,B 0,C 180,E1 -9109.868,E2 -9109.868} C_VEL
LIN {X 0,Y 439.881,Z 638.535,A -85,B 0,C 180,E1 -9113.294,E2 -9113.294} C_VEL
LIN {X 0,Y 440.472,Z 624.704,A -85,B 0,C 180,E1 -9116.681,E2 -9116.681} C_VEL
LIN {X 0,Y 441.157,Z 609.947,A -85,B 0,C 180,E1 -9120.385,E2 -9120.385} C_VEL
LIN {X 0,Y 441.806,Z 596.592,A -85,B 0,C 180,E1 -9123.833,E2 -9123.833} C_VEL
LIN {X 0,Y 442.32,Z 586.279,A -85,B 0,C 180,E1 -9126.573,E2 -9126.573} C_VEL
LIN {X 0,Y 441.774,Z 581.905,A -85,B 0,C 180,E1 -9127.811,E2 -9127.811} C_VEL
LIN {X 0,Y 439.755,Z 571.371,A -85,B 0,C 180,E1 -9130.939,E2 -9130.939} C_VEL
LIN {X 0,Y 439.419,Z 569.752,A -85,B 0,C 180,E1 -9131.502,E2 -9131.502} C_VEL
LIN {X 0,Y 439.406,Z 569.753,A -85,B 0,C 180,E1 -9135.271,E2 -9135.271} C_VEL
LIN {X 0,Y 439.393,Z 569.755,A -85,B 0,C 180,E1 -9138.743,E2 -9138.743} C_VEL
LIN {X 0,Y 439.39,Z 569.753,A -85,B 0,C 180,E1 -9141.606,E2 -9141.606} C_VEL
LIN {X 0,Y 439.406,Z 569.751,A -85,B 0,C 180,E1 -9144.844,E2 -9144.844} C_VEL
LIN {X 0,Y 439.377,Z 569.756,A -85,B 0,C 180,E1 -9148.14,E2 -9148.14} C_VEL
LIN {X 0,Y 439.437,Z 569.746,A -85,B 0,C 180,E1 -9151.598,E2 -9151.598} C_VEL
LIN {X 0,Y 439.41,Z 569.753,A -85,B 0,C 180,E1 -9154.415,E2 -9154.415} C_VEL
LIN {X 0,Y 439.369,Z 569.754,A -85,B 0,C 180,E1 -9157.424,E2 -9157.424} C_VEL
LIN {X 0,Y 439.446,Z 569.747,A -85,B 0,C 180,E1 -9160.663,E2 -9160.663} C_VEL
LIN {X 0,Y 439.467,Z 569.745,A -85,B 0,C 180,E1 -9164.224,E2 -9164.224} C_VEL
LIN {X 0,Y 439.488,Z 569.742,A -85,B 0,C 180,E1 -9168.001,E2 -9168.001} C_VEL
LIN {X 0,Y 439.552,Z 569.732,A -85,B 0,C 180,E1 -9171.726,E2 -9171.726} C_VEL
LIN {X 0,Y 439.625,Z 569.726,A -85,B 0,C 180,E1 -9174.495,E2 -9174.495} C_VEL
LIN {X 0,Y 439.637,Z 569.724,A -85,B 0,C 180,E1 -9178.167,E2 -9178.167} C_VEL
LIN {X 0,Y 439.768,Z 569.707,A -85,B 0,C 180,E1 -9180,E2 -9180} C_VEL
LIN {X 0,Y 439.643,Z 569.722,A -85,B 0,C 180,E1 -9182.748,E2 -9182.748} C_VEL
LIN {X 0,Y 439.622,Z 569.726,A -85,B 0,C 180,E1 -9186.425,E2 -9186.425} C_VEL
LIN {X 0,Y 439.503,Z 569.739,A -85,B 0,C 180,E1 -9189.201,E2 -9189.201} C_VEL
LIN {X 0,Y 439.469,Z 569.743,A -85,B 0,C 180,E1 -9192.937,E2 -9192.937} C_VEL
LIN {X 0,Y 439.45,Z 569.748,A -85,B 0,C 180,E1 -9196.348,E2 -9196.348} C_VEL
LIN {X 0,Y 439.405,Z 569.75,A -85,B 0,C 180,E1 -9199.626,E2 -9199.626} C_VEL
LIN {X 0,Y 439.368,Z 569.757,A -85,B 0,C 180,E1 -9202.575,E2 -9202.575} C_VEL
LIN {X 0,Y 439.407,Z 569.75,A -85,B 0,C 180,E1 -9205.584,E2 -9205.584} C_VEL
LIN {X 0,Y 439.419,Z 569.751,A -85,B 0,C 180,E1 -9208.673,E2 -9208.673} C_VEL
